// TwinCAT 3 PLC project MainControl
// ProgramVersion: 3.1.4023.0
// libraries:
//   Tc2_EtherCAT, * (Beckhoff Automation GmbH)
//   Tc2_SerialCom, * (Beckhoff Automation GmbH)
//   Tc2_Standard, * (Beckhoff Automation GmbH)
//   Tc2_System, * (Beckhoff Automation GmbH)
//   Tc2_Utilities, * (Beckhoff Automation GmbH)
//   Tc3_EventLogger, * (Beckhoff Automation GmbH)
//   Tc3_Module, * (Beckhoff Automation GmbH)
// project tree:
//   DUTs/ ActivationStatus.TcDUT (not stored), GCControllerMode.TcDUT, GuidanceSystemSTM.TcDUT, HighLevelCondition.TcDUT, LEDColor.TcDUT (not stored), LEDMode.TcDUT (not stored), LevitationSystemSTM.TcDUT (not stored), OperationControlCommands.TcDUT (not stored), TGControllerMode.TcDUT (not stored), TopLevelSTM.TcDUT (not stored), ServiceModuleSTM.TcDUT (not stored), SubLevelCondition.TcDUT, XMCCommands.TcDUT
//   DUTs/Interfaces/ ForwardXMCToOperationControl.TcDUT, FromMainControlToOperationControl.TcDUT, FromMainControlToXMC.TcDUT, FromOperationControlToMainControl.TcDUT (not stored), FromXMCToMainControl.TcDUT
//   GVLs/ OperationControlData.TcGVL, Test.TcGVL, XMCData.TcGVL
//   OOPs/ FB_HighLevelSystem.TcPOU, ITF_HighLevelSystem.TcIO, ITF_SubSystem.TcIO (not stored)
//   POUs/ErrorHandling/ FB_SafetyCounter.TcPOU, FB_EventLogging.TcPOU
//   POUs/ FB_LevitationSystem.TcPOU, PRG_ErrorHandling.TcPOU, PRG_MainController.TcPOU, FB_GuidanceSystem.TcPOU, FB_ServiceModule.TcPOU
//   / PlcTask.TcTTO, PlcTask_Fast.TcTTO
//   POUs/Guidance/AccelerationSensor/ AccelerationSensor.TcGVL, FB_SerialComRS232.TcPOU
//   POUs/Guidance/ FB_AccelerationSensor.TcPOU, FB_GuidanceController.TcPOU
//   POUs/Levitation/ FB_EqualizingController.TcPOU, FB_TrajectoryGenerator.TcPOU
//   POUs/ServiceModule/BoxLED/ BoxLED.TcGVL
//   POUs/ServiceModule/DistanceSensor/ DistanceSensor.TcGVL, FB_SerialComRS422.TcPOU
//   POUs/ServiceModule/ FB_BoxLED.TcPOU, FB_DistanceSensor.TcPOU, FB_RGBLED.TcPOU
//   POUs/ServiceModule/RGBLED/ RGBLED.TcGVL
// real-time tasks:
//   TASK PlcTask: cycle T#1ms, priority 20, ADS port 351
//   TASK PlcTask_Fast: cycle T#1ms, priority 19, ADS port 350
// I/O:
//   DEVICE Gerät 3 (EtherCAT) (disabled), AmsNetId 10.183.66.136.4.1
//     Klemme 1 (EK1100) [EK1100 EtherCAT-Koppler (2A E-Bus)]
//       Klemme 2 (EL6021) [EL6021 Schnittstelle (RS422/485)]
//       Klemme 3 (EL6001) [EL6001 Schnittstelle (RS232)]
//       Klemme 4 (EL6001) [EL6001 Schnittstelle (RS232)]
//       Klemme 5 (EL2564) [EL2564 4 K. LED-Ausgang, 5...48 V DC, 4 A, RGBW]
//       Klemme 6 (EL9011) [EL9011 Endklemme]
//   DEVICE Gerät 4 (EtherCAT Slave) (disabled), AmsNetId 10.183.66.136.5.255
// variable links:
//   MainControl/MainControl Instance <-> Device 3 (EtherCAT)/Term 1 (EK1100)/Term 2 (EL6021)
//     PlcTask Inputs/DistanceSensor.stEL6021In @bit {16..184 step 8} <-> COM TxPDO-Map Inputs/Data In {0..21}  (22 links)
//     PlcTask Inputs/DistanceSensor.stEL6021In <-> COM TxPDO-Map Inputs/Status
//     PlcTask Outputs/DistanceSensor.stEL6021Out <-> COM RxPDO-Map Outputs/Ctrl
//     PlcTask Outputs/DistanceSensor.stEL6021Out @bit {16..184 step 8} <-> COM RxPDO-Map Outputs/Data Out {0..21}  (22 links)
//   MainControl/MainControl Instance <-> Device 3 (EtherCAT)/Term 1 (EK1100)/Term 3 (EL6001)
//     PlcTask Inputs/AccelerationSensor.stEL6001InIMU1 @bit {16..184 step 8} <-> COM Inputs/Data In {0..21}  (22 links)
//     PlcTask Inputs/AccelerationSensor.stEL6001InIMU1 <-> COM Inputs/Status
//     PlcTask Outputs/AccelerationSensor.stEL6001OutIMU1 <-> COM Outputs/Ctrl
//     PlcTask Outputs/AccelerationSensor.stEL6001OutIMU1 @bit {16..184 step 8} <-> COM Outputs/Data Out {0..21}  (22 links)
//   MainControl/MainControl Instance <-> Device 3 (EtherCAT)/Term 1 (EK1100)/Term 4 (EL6001)
//     PlcTask Inputs/AccelerationSensor.stEL6001InIMU2 @bit {16..184 step 8} <-> COM Inputs/Data In {0..21}  (22 links)
//     PlcTask Inputs/AccelerationSensor.stEL6001InIMU2 <-> COM Inputs/Status
//     PlcTask Outputs/AccelerationSensor.stEL6001OutIMU2 <-> COM Outputs/Ctrl
//     PlcTask Outputs/AccelerationSensor.stEL6001OutIMU2 @bit {16..184 step 8} <-> COM Outputs/Data Out {0..21}  (22 links)
//   MainControl/MainControl Instance <-> Device 3 (EtherCAT)/Term 1 (EK1100)/Term 5 (EL2564)
//     PlcTask Inputs/BoxLED.bBoxGreenError <-> PWM Inputs Channel 4/Status/Error
//     PlcTask Inputs/BoxLED.bBoxGreenWarning <-> PWM Inputs Channel 4/Status/Warning
//     PlcTask Outputs/BoxLED.nBoxGreen <-> PWM Outputs Channel 4/PWM output
//   MainControl/MainControl Instance <-> Device 4 (EtherCAT Slave)
//     PlcTask Inputs/OperationControlData.stFromOCToMC <-> Inputs/FromOCToMC
//     PlcTask Outputs/OperationControlData.stForwardXMC{1..4}ToOC <-> Outputs/ForwardXMC{1..4}ToOC  (4 links)
//     PlcTask Outputs/OperationControlData.stFromMCToOC <-> Outputs/FromMCToOC

CONFIGURATION MainControl
    RESOURCE PLC ON TwinCAT3
        TASK PlcTask(INTERVAL := T#1ms, PRIORITY := 20);
        TASK PlcTask_Fast(INTERVAL := T#1ms, PRIORITY := 19);
        PROGRAM PRG_ErrorHandling WITH PlcTask : PRG_ErrorHandling;
        PROGRAM PRG_MainController WITH PlcTask : PRG_MainController;
        PROGRAM PRG_ErrorHandling WITH PlcTask_Fast : PRG_ErrorHandling;
    END_RESOURCE
END_CONFIGURATION

// ---- DUTs/GCControllerMode.TcDUT
{attribute 'qualified_only'}
{attribute 'strict'}
TYPE GCControllerMode :
(
	CurrentControlled,
	ForceControlled
);
END_TYPE

// ---- DUTs/GuidanceSystemSTM.TcDUT
{attribute 'qualified_only'}
{attribute 'strict'}
TYPE GuidanceSystemSTM :
(
	Idling,
	PreRunning,
	Running,
	PostRunning
);
END_TYPE

// ---- DUTs/HighLevelCondition.TcDUT
{attribute 'qualified_only'}
{attribute 'strict'}
TYPE HighLevelCondition :
(
	INIT,
	RUN,
	SLEEP
);
END_TYPE

// ---- DUTs/Interfaces/ForwardXMCToOperationControl.TcDUT
TYPE ForwardXMCToOperationControl :
STRUCT
	MO_origE_State							:	USINT			;
	MO_origE_LoggingCounterIn               :	USINT			;
	MO_origE_LoggingCounterSize             :	USINT			;
	MO_origE_LoggingCounterBuf0             :	BYTE			;
	MO_origE_LoggingCounterBuf1             :	BYTE			;
	MO_origE_LoggingCounterBuf2             :	BYTE			;
	MO_origE_LoggingCounterBuf3             :	BYTE			;
	MO_origE_LoggingCounterBuf4             :	BYTE			;
	MO_origE_LoggingCounterBuf5             :	BYTE			;
	MO_origE_LoggingCounterBuf6             :	BYTE			;
	MO_origE_LoggingCounterBuf7             :	BYTE			;
	MO_origE_LoggingCounterBuf8             :	BYTE			;
	MO_origE_LoggingCounterBuf9             :	BYTE			;
	MO_origE_SafetyCounter                  :	UDINT			;
	MO_origE_Timestamp                      :	UDINT			;
	MO_origE_WarnBits                       :	ULINT			;
	MO_origE_ErrBits                        :	ULINT			;
	MO_origE_DistanceLevitationFiltered     :	REAL			;
	MO_origE_DistanceGuidanceFiltered       :	REAL			;
	MO_origE_DistanceRawLev11               :	REAL			;
	MO_origE_DistanceRawLev12               :	REAL			;
	MO_origE_DistanceRawLev21               :	REAL			;
	MO_origE_DistanceRawLev22               :	REAL			;
	MO_origE_DistanceRawGuid11              :	REAL			;
	MO_origE_DistanceRawGuid12              :	REAL			;
	MO_origE_IMUX                           :	REAL			;
	MO_origE_IMUY                           :	REAL			;
	MO_origE_IMUZ                           :	REAL			;
	MO_origE_VelocityZFiltered              :	REAL			;
	MO_origE_TemperatureBox                 :	REAL			;
	MO_origE_TemperatureLev0                :	REAL			;
	MO_origE_TemperatureLev1                :	REAL			;
	MO_origE_TemperatureGuid                :	REAL			;
	MO_origE_PressureBox                    :	REAL			;
	MO_origE_CurrentLev                     :	DINT			;
	MO_origE_CurrentGuid                    :	DINT			;
	MO_origE_GuidEstimatedFlux0             :	ARRAY [0..1] OF REAL			;
	MO_origE_GuidEstimatedFlux1             :	ARRAY [0..1] OF REAL			;
	MO_origE_GuidEstimatedCurrent           :	REAL			;
	MO_origE_GuidEstimatedResistance        :	REAL			;
	MO_origE_GuidIntegratedControlError     :	REAL			;
	MO_origE_GuidReferenceVoltage           :	REAL			;
	MO_origE_LevEstimatedFlux0              :	ARRAY [0..1] OF REAL			;
	MO_origE_LevEstimatedFlux1              :	ARRAY [0..1] OF REAL			;
	MO_origE_LevEstimatedCurrent            :	REAL			;
	MO_origE_LevEstimatedResistance         :	REAL			;
	MO_origE_LevIntegratedControlError      :	REAL			;
	MO_origE_LevReferenceVoltage            :	REAL			;
END_STRUCT
END_TYPE

// ---- DUTs/Interfaces/FromMainControlToOperationControl.TcDUT
TYPE FromMainControlToOperationControl :
STRUCT
		//MainController
		MO_origM_State 							: USINT		;
		MO_origM_WarnBits 						: ULINT		;
		MO_origM_ErrBits 						: ULINT		;
		MO_origM_SafetyCounter 					: UDINT		;
		MO_origM_ShutdownFinished 				: BIT		;
		//ServiceModule                 		
		MO_origM_DistanceServiceModule 			: REAL		;
		
		//LevitationSystem
		MO_origM_ECOutputDistanceXMC1 			: REAL		;
		MO_origM_ECOutputDistanceXMC2 			: REAL		;
		MO_origM_ECOutputDistanceXMC3 			: REAL		;
		MO_origM_ECOutputDistanceXMC4 			: REAL		;
		MO_origM_TGOutputLevDistanceXMC1 		: REAL		;
		MO_origM_TGOutputLevDistanceXMC2 		: REAL		;
		MO_origM_TGOutputLevDistanceXMC3 		: REAL		;
		MO_origM_TGOutputLevDistanceXMC4 		: REAL		;
		MO_origM_TGOutputLevVelocityXMC1 		: REAL		;
		MO_origM_TGOutputLevVelocityXMC2 		: REAL		;
		MO_origM_TGOutputLevVelocityXMC3 		: REAL		;
		MO_origM_TGOutputLevVelocityXMC4 		: REAL		;
		MO_origM_TGOutputLevAccelerationXMC1 	: REAL		;
		MO_origM_TGOutputLevAccelerationXMC2 	: REAL		;
		MO_origM_TGOutputLevAccelerationXMC3 	: REAL		;
		MO_origM_TGOutputLevAccelerationXMC4 	: REAL		;
		MO_origM_TGOutputLevCurrentXMC1 		: REAL		;
		MO_origM_TGOutputLevCurrentXMC2 		: REAL		;
		MO_origM_TGOutputLevCurrentXMC3 		: REAL		;
		MO_origM_TGOutputLevCurrentXMC4 		: REAL		;
		MO_origM_TGOutputLevVoltageXMC1 		: REAL		;
		MO_origM_TGOutputLevVoltageXMC2 		: REAL		;
		MO_origM_TGOutputLevVoltageXMC3 		: REAL		;
		MO_origM_TGOutputLevVoltageXMC4 		: REAL		;
		MO_origM_TGOutputLevForceXMC1 			: REAL		;
		MO_origM_TGOutputLevForceXMC2 			: REAL		;
		MO_origM_TGOutputLevForceXMC3 			: REAL		;
		MO_origM_TGOutputLevForceXMC4 			: REAL		;
		
		//GuidanceSystem
		MO_origM_GuidanceIMUX0 					: REAL		;
		MO_origM_GuidanceIMUX1 					: REAL		;
		MO_origM_GuidanceIMUY0 					: REAL		;
		MO_origM_GuidanceIMUY1 					: REAL		;
		MO_origM_GuidanceIMUZ0 					: REAL		;
		MO_origM_GuidanceIMUZ1 					: REAL		;
		MO_origM_GCOutputGuidCurrentXMC1 		: REAL		;
		MO_origM_GCOutputGuidCurrentXMC2 		: REAL		;
		MO_origM_GCOutputGuidCurrentXMC3 		: REAL		;
		MO_origM_GCOutputGuidCurrentXMC4 		: REAL		;
		MO_origM_GCOutputGuidVoltageXMC1 		: REAL		;
		MO_origM_GCOutputGuidVoltageXMC2 		: REAL		;
		MO_origM_GCOutputGuidVoltageXMC3 		: REAL		;
		MO_origM_GCOutputGuidVoltageXMC4 		: REAL		;
		MO_origM_GCOutputGuidForceXMC1 			: REAL		;
		MO_origM_GCOutputGuidForceXMC2 			: REAL		;
		MO_origM_GCOutputGuidForceXMC3 			: REAL		;
		MO_origM_GCOutputGuidForceXMC4 			: REAL		;
END_STRUCT
END_TYPE

// ---- DUTs/Interfaces/FromMainControlToXMC.TcDUT
TYPE FromMainControlToXMC :
STRUCT
	ME_origM_StartOperational						:	BIT		;
	ME_origM_StopOperational                        :	BIT    	;
	ME_origM_AckError                               :	BIT    	;
	ME_origG_Logging_CounterOut                     :	USINT   ;
	ME_origM_SafetyCounter                          :	UDINT   ;
	ME_origM_DesiredGuidCurrent                     :	REAL    ;
	ME_origM_DesiredGuidForce                       :	REAL    ;
	ME_origM_DesiredGuidVoltage                     :	REAL    ;
	ME_origM_DesiredLevDistance                     :	REAL    ;
	ME_origM_DesiredLevVelocity                     :	REAL    ;
	ME_origM_DesiredLevAcceleration                 :	REAL    ;
	ME_origM_DesiredLevForce                        :	REAL    ;
	ME_origM_DesiredLevCurrent                      :	REAL    ;
	ME_origM_DesiredLevVoltage                      :	REAL    ;
	ME_origM_DebugPWMLev                            :	INT     ;
	ME_origM_DebugPWMGuid                           :	INT     ;
	ME_origM_DebugSel                               :	USINT   ;
	ME_origG_GuidControlOption                      :	USINT   ;
	ME_origG_LevControlOption                       :	USINT   ;
	ME_origG_EnableGuidController                   :	BIT    	;
	ME_origM_GuidEnableCurrentController            :	BIT    	;
	ME_origM_GuidEnableIControl                     :	BIT    	;
	ME_origM_GuidEnablePControl                     :	BIT    	;
	ME_origM_LevEnableCurrentController             :	BIT    	;
	ME_origM_LevEnableIControl                      :	BIT    	;
	ME_origM_LevEnablePControl                      :	BIT    	;
END_STRUCT
END_TYPE

// ---- DUTs/Interfaces/FromXMCToMainControl.TcDUT
TYPE FromXMCToMainControl :
STRUCT
	EM_origE_State							:	USINT			;
	EM_origE_LoggingCounterIn               :	USINT			;
	EM_origE_LoggingCounterSize             :	USINT			;
	EM_origE_LoggingCounterBuf0             :	BYTE			;
	EM_origE_LoggingCounterBuf1             :	BYTE			;
	EM_origE_LoggingCounterBuf2             :	BYTE			;
	EM_origE_LoggingCounterBuf3             :	BYTE			;
	EM_origE_LoggingCounterBuf4             :	BYTE			;
	EM_origE_LoggingCounterBuf5             :	BYTE			;
	EM_origE_LoggingCounterBuf6             :	BYTE			;
	EM_origE_LoggingCounterBuf7             :	BYTE			;
	EM_origE_LoggingCounterBuf8             :	BYTE			;
	EM_origE_LoggingCounterBuf9             :	BYTE			;
	EM_origE_SafetyCounter                  :	UDINT			;
	EM_origE_Timestamp                      :	UDINT			;
	EM_origE_WarnBits                       :	ULINT			;
	EM_origE_ErrBits                        :	ULINT			;
	EM_origE_DistanceLevitationFiltered     :	REAL			;
	EM_origE_DistanceGuidanceFiltered       :	REAL			;
	EM_origE_DistanceRawLev11               :	REAL			;
	EM_origE_DistanceRawLev12               :	REAL			;
	EM_origE_DistanceRawLev21               :	REAL			;
	EM_origE_DistanceRawLev22               :	REAL			;
	EM_origE_DistanceRawGuid11              :	REAL			;
	EM_origE_DistanceRawGuid12              :	REAL			;
	EM_origE_IMUX                           :	REAL			;
	EM_origE_IMUY                           :	REAL			;
	EM_origE_IMUZ                           :	REAL			;
	EM_origE_VelocityZFiltered              :	REAL			;
	EM_origE_TemperatureBox                 :	REAL			;
	EM_origE_TemperatureLev0                :	REAL			;
	EM_origE_TemperatureLev1                :	REAL			;
	EM_origE_TemperatureGuid                :	REAL			;
	EM_origE_PressureBox                    :	REAL			;
	EM_origE_CurrentLev                     :	DINT			;
	EM_origE_CurrentGuid                    :	DINT			;
	EM_origE_GuidEstimatedFlux0             :	ARRAY [0..1] OF REAL;
	EM_origE_GuidEstimatedFlux1             :	ARRAY [0..1] OF REAL			;
	EM_origE_GuidEstimatedCurrent           :	REAL			;
	EM_origE_GuidEstimatedResistance        :	REAL			;
	EM_origE_GuidIntegratedControlError     :	REAL			;
	EM_origE_GuidReferenceVoltage           :	REAL			;
	EM_origE_LevEstimatedFlux0              :	ARRAY [0..1] OF REAL			;
	EM_origE_LevEstimatedFlux1              :	ARRAY [0..1] OF REAL			;
	EM_origE_LevEstimatedCurrent            :	REAL			;
	EM_origE_LevEstimatedResistance         :	REAL			;
	EM_origE_LevIntegratedControlError      :	REAL			;
	EM_origE_LevReferenceVoltage            :	REAL			;
END_STRUCT
END_TYPE

// ---- DUTs/SubLevelCondition.TcDUT
{attribute 'qualified_only'}
{attribute 'strict'}
TYPE SubLevelCondition :
(
	ERROR,
	RUN
);
END_TYPE

// ---- DUTs/XMCCommands.TcDUT
TYPE XMCCommands :
STRUCT
	//MainController
	nSafetyCounterXMC1 			: UDINT	;
	nSafetyCounterXMC2 			: UDINT	;
	nSafetyCounterXMC3 			: UDINT	;
	nSafetyCounterXMC4 			: UDINT	;
	nStateXMC1					: USINT	;
	nStateXMC2					: USINT	;
	nStateXMC3					: USINT	;
	nStateXMC4					: USINT	;
	
	//Outputs
	bStartOperational : BOOL;
	bStopOperational	: BOOL;
	bAckError			: BOOL;
	nDebugPWMSel		: USINT;
	nDebugPWMLev		: INT;
	nDebugPWMGuid		: INT;
END_STRUCT
END_TYPE

// ---- GVLs/OperationControlData.TcGVL
{attribute 'qualified_only'}
VAR_GLOBAL
	stFromOCToMC 			AT %I* : FromOperationControlToMainControl;
	
	stFromMCToOC 			AT %Q* : FromMainControlToOperationControl;
	stForwardXMC1ToOC 		AT %Q* : ForwardXMCToOperationControl;
	stForwardXMC2ToOC 		AT %Q* : ForwardXMCToOperationControl;
	stForwardXMC3ToOC 		AT %Q* : ForwardXMCToOperationControl;
	stForwardXMC4ToOC 		AT %Q* : ForwardXMCToOperationControl;
END_VAR

// ---- GVLs/Test.TcGVL
{attribute 'qualified_only'}
VAR_GLOBAL
	nTest AT %Q* : INT;
END_VAR

// ---- GVLs/XMCData.TcGVL
{attribute 'qualified_only'}
VAR_GLOBAL
	stFromXMC1ToMC 			AT %I* : FromXMCToMainControl;
	stFromXMC2ToMC 			AT %I* : FromXMCToMainControl;
	stFromXMC3ToMC 			AT %I* : FromXMCToMainControl;
	stFromXMC4ToMC 			AT %I* : FromXMCToMainControl;
	
	stFromMCToXMC1			AT %Q* : FromMainControlToXMC;
	stFromMCToXMC2			AT %Q* : FromMainControlToXMC;
	stFromMCToXMC3			AT %Q* : FromMainControlToXMC;
	stFromMCToXMC4			AT %Q* : FromMainControlToXMC;
END_VAR

// ---- POUs/Guidance/AccelerationSensor/AccelerationSensor.TcGVL
VAR_GLOBAL
	stEL6001InIMU1 AT %I*	: EL6inData22B;		//**To EL6001 Inputs incl. Status (Clamp 3)**
	stEL6001OutIMU1 AT %Q*	: EL6outData22B;	//**To EL6001 Outputs incl. Ctrl (Clamp 3)**
	
	stEL6001InIMU2 AT %I*	: EL6inData22B;		//**To EL6001 Inputs incl. Status (Clamp 4)**
	stEL6001OutIMU2 AT %Q*	: EL6outData22B;	//**To EL6001 Outputs incl. Ctrl (Clamp 4)** 
END_VAR

// ---- POUs/ServiceModule/BoxLED/BoxLED.TcGVL
{attribute 'qualified_only'}
VAR_GLOBAL
	nBoxGreen AT %Q* : INT;					//**To EL2564 PWM Outputs Channel 4 (PWM output)**
	
	bBoxGreenError AT %I* : BOOL;				//**To EL2564 PWM Inputs Channel 4 (Status -> Error)**
	bBoxGreenWarning AT %I* : BOOL;			//**To EL2564 PWM Inputs Channel 4 (Status -> Warning)**
END_VAR

// ---- POUs/ServiceModule/DistanceSensor/DistanceSensor.TcGVL
{attribute 'qualified_only'}
VAR_GLOBAL
	stEL6021In  AT %I*	: EL6inData22B;		//**To EL6021 Inputs**
	stEL6021Out AT %Q*	: EL6outData22B;	//**To EL6021 Outputs**
END_VAR

// ---- POUs/ServiceModule/RGBLED/RGBLED.TcGVL
{attribute 'qualified_only'}
VAR_GLOBAL
	nRed AT %Q* : INT;				//**To EL2564 PWM Outputs Channel 1 (PWM output)**
	nGreen AT %Q* : INT;			//**To EL2564 PWM Outputs Channel 2 (PWM output)**
	nBlue AT %Q* : INT;				//**To EL2564 PWM Outputs Channel 3 (PWM output)**
	
	bRedError AT %I* : BOOL;		//**To EL2564 PWM Inputs Channel 1 (Status -> Error)**
	bRedWarning AT %I* : BOOL;		//**To EL2564 PWM Inputs Channel 1 (Status -> Warning)**
	bGreenError AT %I* : BOOL;		//**To EL2564 PWM Inputs Channel 2 (Status -> Error)**
	bGreenWarning AT %I* : BOOL;	//**To EL2564 PWM Inputs Channel 2 (Status -> Warning)**
	bBlueError AT %I* : BOOL;		//**To EL2564 PWM Inputs Channel 3 (Status -> Error)**
	bBlueWarning AT %I* : BOOL;		//**To EL2564 PWM Inputs Channel 3 (Status -> Warning)**
END_VAR

// ---- OOPs/ITF_HighLevelSystem.TcIO
INTERFACE ITF_HighLevelSystem

PROPERTY PUBLIC eCondition : HighLevelCondition
GET
END_GET
END_PROPERTY

PROPERTY PUBLIC nErrorID : UDINT
GET
END_GET
END_PROPERTY

END_INTERFACE

// ---- POUs/PRG_ErrorHandling.TcPOU
PROGRAM PRG_ErrorHandling
VAR
	nErrorBits 						: ULINT;
	nWarningBits 					: ULINT;
	
	fbStartUpTimer 					: TON := (PT := tStartUpTime);
	fbShutdownTimer					: TON := (PT := tShutdownTime);
	bStartUpCheck 					: BOOL;
	bErrorInStartUp 				: BOOL;
	bErrorInReady 					: BOOL;
	bErrorInOperational 			: BOOL;
	bErrorInShutdown 				: BOOL;
	bGoToError						: BOOL;
	bAllErrorsAcknowledged 			: BOOL;
	
	fbEventLogging 					: FB_EventLogging;
	aSetEventCounterToZero 			: ARRAY [0..nNumberOfWarnings + nNumberOfErrors + nNumberOfInfos - 1] OF USINT;
	n 								: USINT;
	
	fbSafetyCounter 				: FB_SafetyCounter;
	
	bDebugMode 						: BOOL;
	nTestMode						: USINT := 63;  //*see test modes table in README*
END_VAR
VAR CONSTANT
	tStartUpTime 					: TIME := T#10S;
	tSafetyCounterTimeout 			: TIME := T#5S;
	tShutdownTime					: TIME := T#30S;
	
	nNumberOfWarnings 				: USINT := 52;			//*set the number of Warnings here*
	nNumberOfErrors 				: USINT := 6;			//*set the number of Errors here*
	nNumberOfInfos					: USINT := 4;			//*set the number of Infos here*
END_VAR

doSetWarningBits(	nErrorIDServiceModule := PRG_MainController.fbServiceModule.nErrorID,
					nErrorIDLevitationSystem := PRG_MainController.fbLevitationSystem.nErrorID,
					nErrorIDGuidanceSystem := PRG_MainController.fbGuidanceSystem.nErrorID,
					nErrorIDMainController := PRG_ErrorHandling.fbSafetyCounter.nErrorID);
					
doSetErrorBits(		nErrorIDServiceModule := PRG_MainController.fbServiceModule.nErrorID,
					nErrorIDLevitationSystem := PRG_MainController.fbLevitationSystem.nErrorID,
					nErrorIDGuidanceSystem := PRG_MainController.fbGuidanceSystem.nErrorID,
					nErrorIDMainController := PRG_ErrorHandling.fbSafetyCounter.nErrorID);

doCheckErrorStates();

fbSafetyCounter();
fbEventLogging();

IF bDebugMode THEN
	nErrorBits := 0;
END_IF

							
CASE PRG_MainController.eState OF
	TopLevelSTM.STARTUP:
		bAllErrorsAcknowledged := FALSE;
		
		IF NOT bDebugMode AND NOT nTestMode.1 THEN
			doStartUpCheck(	eConditionServiceModule := PRG_MainController.fbServiceModule.eCondition,
							eConditionLevitationSystem := PRG_MainController.fbLevitationSystem.eCondition,
							eConditionGuidanceSystem := PRG_MainController.fbGuidanceSystem.eCondition);
		ELSE
			bStartUpCheck := TRUE;
		END_IF	
										
	TopLevelSTM.READY:
		fbShutdownTimer(IN:=FALSE);
		IF nErrorBits <> 0 THEN
			bErrorInReady := TRUE;
		ELSE
			bErrorInReady := FALSE;
		END_IF
		
	TopLevelSTM.OPERATIONAL:
		IF nErrorBits <> 0 THEN
			bErrorInOperational := TRUE;
		ELSE
			bErrorInOperational := FALSE;
		END_IF
		
	TopLevelSTM.SHUTDOWN:
		fbShutdownTimer(IN:=TRUE);
		IF NOT bErrorInOperational THEN
			IF nErrorBits <> 0 THEN
				bErrorInShutdown := TRUE;
			ELSE
				bErrorInShutdown := FALSE;
			END_IF
		END_IF
		
	TopLevelSTM.ERROR:
		IF PRG_MainController.stOperationControlCommands.bAckError THEN
			
			//Reset WarningBits and ErrorBits
			nWarningBits := 0;
			nErrorBits := 0;
			
			//Reset Event Logging
			FOR n := 0 TO nNumberOfWarnings + nNumberOfErrors + nNumberOfInfos -1 DO
				aSetEventCounterToZero[n] := 0;
			END_FOR
			fbEventLogging.aEventCounter := aSetEventCounterToZero;
			
			//ResetSafetyCounter
			fbSafetyCounter(bReset := TRUE);
			fbSafetyCounter.bReset := FALSE;
			
			//Acknowledge
			bErrorInStartUp := FALSE;
			bErrorInReady := FALSE;
			bErrorInOperational := FALSE;
			bErrorInShutdown := FALSE;
			bAllErrorsAcknowledged := TRUE;
		END_IF
END_CASE

METHOD PRIVATE doCheckErrorStates
IF PRG_MainController.stXMCCommands.nStateXMC1 = 3 OR PRG_MainController.stXMCCommands.nStateXMC2 = 3 OR PRG_MainController.stXMCCommands.nStateXMC3 = 3 OR PRG_MainController.stXMCCommands.nStateXMC4 = 3 OR PRG_MainController.stOperationControlCommands.bGoToError THEN
	bGoToError := TRUE;
ELSE
	bGoToError := FALSE;
END_IF
END_METHOD

METHOD PRIVATE doSetErrorBits
VAR_INPUT
	nErrorIDServiceModule : UDINT;
	nErrorIDLevitationSystem : UDINT;
	nErrorIDGuidanceSystem : UDINT;
	nErrorIDMainController : UDINT;
END_VAR
IF PRG_MainController.fbServiceModule.eActivationStatus = ActivationStatus.Disabled THEN
	nErrorIDServiceModule := 0;
END_IF
IF PRG_MainController.fbLevitationSystem.eActivationStatus = ActivationStatus.Disabled THEN
	nErrorIDLevitationSystem := 0;
	nErrorIDMainController.1 := 0;
	nErrorIDMainController.2 := 0;
	nErrorIDMainController.3 := 0;
	nErrorIDMainController.4 := 0;
END_IF
IF PRG_MainController.fbGuidanceSystem.eActivationStatus = ActivationStatus.Disabled THEN
	nErrorIDGuidanceSystem := 0;
	nErrorIDMainController.1 := 0;
	nErrorIDMainController.2 := 0;
	nErrorIDMainController.3 := 0;
	nErrorIDMainController.4 := 0;
END_IF


//ServiceModule

//LevitationSystem

//GuidanceSystem
		
//MainController
nErrorBits.0 := nErrorIDMainController.0;
nErrorBits.1 := nErrorIDMainController.1;
nErrorBits.2 := nErrorIDMainController.2;
nErrorBits.3 := nErrorIDMainController.3;
nErrorBits.4 := nErrorIDMainController.4;
nErrorBits.5 := nErrorIDMainController.5;
END_METHOD

METHOD PRIVATE doSetWarningBits
VAR_INPUT
	nErrorIDServiceModule : UDINT;
	nErrorIDLevitationSystem : UDINT;
	nErrorIDGuidanceSystem : UDINT;
	nErrorIDMainController : UDINT;
END_VAR
IF PRG_MainController.fbServiceModule.eActivationStatus = ActivationStatus.Disabled THEN
	nErrorIDServiceModule := 0;
END_IF
IF PRG_MainController.fbLevitationSystem.eActivationStatus = ActivationStatus.Disabled THEN
	nErrorIDLevitationSystem := 0;
END_IF
IF PRG_MainController.fbGuidanceSystem.eActivationStatus = ActivationStatus.Disabled THEN
	nErrorIDGuidanceSystem := 0;
END_IF

//ServiceModule
nWarningBits.0 := nErrorIDServiceModule.0;
nWarningBits.1 := nErrorIDServiceModule.1;
nWarningBits.2 := nErrorIDServiceModule.2;
nWarningBits.3 := nErrorIDServiceModule.3;
nWarningBits.4 := nErrorIDServiceModule.4;
nWarningBits.5 := nErrorIDServiceModule.5;
nWarningBits.6 := nErrorIDServiceModule.6;
nWarningBits.7 := nErrorIDServiceModule.7;
nWarningBits.8 := nErrorIDServiceModule.8;
nWarningBits.9 := nErrorIDServiceModule.9;

//LevitationSystem
nWarningBits.10 := nErrorIDLevitationSystem.0;
nWarningBits.11 := nErrorIDLevitationSystem.1;
nWarningBits.12 := nErrorIDLevitationSystem.2;
nWarningBits.13 := nErrorIDLevitationSystem.3;
nWarningBits.14 := nErrorIDLevitationSystem.4;
nWarningBits.15 := nErrorIDLevitationSystem.5;
nWarningBits.16 := nErrorIDLevitationSystem.6;
nWarningBits.17 := nErrorIDLevitationSystem.7;
nWarningBits.18 := nErrorIDLevitationSystem.8;
nWarningBits.19 := nErrorIDLevitationSystem.9;
nWarningBits.20 := nErrorIDLevitationSystem.10;
nWarningBits.21 := nErrorIDLevitationSystem.11;
nWarningBits.22 := nErrorIDLevitationSystem.12;
nWarningBits.23 := nErrorIDLevitationSystem.13;
nWarningBits.24 := nErrorIDLevitationSystem.14;
nWarningBits.25 := nErrorIDLevitationSystem.15;
nWarningBits.26 := nErrorIDLevitationSystem.16;
nWarningBits.27 := nErrorIDLevitationSystem.17;
nWarningBits.28 := nErrorIDLevitationSystem.18;
nWarningBits.29 := nErrorIDLevitationSystem.19;
nWarningBits.30 := nErrorIDLevitationSystem.20;
nWarningBits.31 := nErrorIDLevitationSystem.21;
nWarningBits.32 := nErrorIDLevitationSystem.22;
nWarningBits.33 := nErrorIDLevitationSystem.23;
nWarningBits.34 := nErrorIDLevitationSystem.24;
nWarningBits.35 := nErrorIDLevitationSystem.25;


//GuidanceSystem
nWarningBits.36 := nErrorIDGuidanceSystem.0;
nWarningBits.37 := nErrorIDGuidanceSystem.1;
nWarningBits.38 := nErrorIDGuidanceSystem.2;
nWarningBits.39 := nErrorIDGuidanceSystem.3;
nWarningBits.40 := nErrorIDGuidanceSystem.4;
nWarningBits.41 := nErrorIDGuidanceSystem.5;
nWarningBits.42 := nErrorIDGuidanceSystem.6;
nWarningBits.43 := nErrorIDGuidanceSystem.7;
nWarningBits.44 := nErrorIDGuidanceSystem.8;
nWarningBits.45 := nErrorIDGuidanceSystem.9;
nWarningBits.46 := nErrorIDGuidanceSystem.10;
nWarningBits.47 := nErrorIDGuidanceSystem.11;
nWarningBits.48 := nErrorIDGuidanceSystem.12;
nWarningBits.49 := nErrorIDGuidanceSystem.13;
nWarningBits.50 := nErrorIDGuidanceSystem.14;
nWarningBits.51 := nErrorIDGuidanceSystem.15;

//MainController
END_METHOD

METHOD PRIVATE doStartUpCheck
VAR_INPUT
	eConditionServiceModule : HighLevelCondition;
	eConditionLevitationSystem : HighLevelCondition;
	eConditionGuidanceSystem : HighLevelCondition;
END_VAR
IF PRG_MainController.stOperationControlCommands.nOperationMode <> 7 THEN
	IF (eConditionServiceModule = HighLevelCondition.RUN OR eConditionServiceModule = HighLevelCondition.SLEEP) AND (eConditionLevitationSystem = HighLevelCondition.RUN OR eConditionLevitationSystem = HighLevelCondition.SLEEP) AND (eConditionGuidanceSystem = HighLevelCondition.RUN OR eConditionGuidanceSystem = HighLevelCondition.SLEEP) AND NOT (eConditionServiceModule = HighLevelCondition.SLEEP AND eConditionLevitationSystem = HighLevelCondition.SLEEP AND eConditionGuidanceSystem = HighLevelCondition.SLEEP) THEN
		fbStartUpTimer(IN := FALSE);
		bStartUpCheck := TRUE;
	ELSE
		fbStartUpTimer(IN := TRUE);
		IF fbStartUpTimer.Q THEN
			fbStartUpTimer(IN := FALSE);
			bErrorInStartUp := TRUE;
			bStartUpCheck := FALSE;
		ELSE
			bStartUpCheck := FALSE;
		END_IF
	END_IF
ELSE
		fbStartUpTimer(IN := TRUE);
		IF fbStartUpTimer.Q THEN
			fbStartUpTimer(IN := FALSE);
			bErrorInStartUp := TRUE;
			bStartUpCheck := FALSE;
		ELSE
			bStartUpCheck := FALSE;
		END_IF
END_IF
END_METHOD

END_PROGRAM

// ---- POUs/ErrorHandling/FB_EventLogging.TcPOU
FUNCTION_BLOCK FB_EventLogging
VAR
	fbEventMessage : FB_TcMessage;
	fbEventLogger : FB_TcEventLogger;
	fbCsvExport : FB_TcEventCsvExportSettings;
	fbCsvClear : FB_TcClearLoggedEventsSettings;

	
	n : USINT;
	aCounterID : ARRAY [0..PRG_ErrorHandling.nNumberOfWarnings + PRG_ErrorHandling.nNumberOfErrors + PRG_ErrorHandling.nNumberOfInfos - 1] OF USINT;
	aWarningArray : ARRAY [0..PRG_ErrorHandling.nNumberOfWarnings-1] OF BOOL;
	aWarningMessagesAsStrings : ARRAY [0..PRG_ErrorHandling.nNumberOfWarnings-1] OF STRING;
	aErrorArray : ARRAY [0..PRG_ErrorHandling.nNumberOfErrors-1] OF BOOL;
	aErrorMessagesAsStrings : ARRAY [0..PRG_ErrorHandling.nNumberOfErrors-1] OF STRING;
	aInfoArray : ARRAY [0..PRG_ErrorHandling.nNumberOfInfos-1] OF BOOL;
	aInfoMessagesAsStrings : ARRAY [0..PRG_ErrorHandling.nNumberOfInfos - 1] OF STRING;
	eMainControllerState : TopLevelSTM;
	sMainControllerStateAsString : STRING;
	
	bClearLoggedEvents : BOOL;
	fbExportTimer : TON;
END_VAR
VAR CONSTANT
	nCounterMax : USINT := 255; //max value for USINT data type
	nCounterReset : USINT := 2;
END_VAR

//CSV-Export
fbExportTimer(IN:=TRUE, PT:=T#5S);
IF fbExportTimer.Q THEN
	fbEventLogger.ExportLoggedEvents(sFileName:='C:\Users\Administrator\Desktop\Log.csv', ipExportSettings := fbCsvExport);
	fbExportTimer(IN := FALSE);
END_IF
//CSV-Clear
IF bClearLoggedEvents THEN
	fbEventLogger.ClearLoggedEvents(ipClearSettings:=fbCsvClear);	
END_IF

//TransitionLogging
sMainControllerStateAsString := TO_STRING(PRG_MainController.eState);
IF eMainControllerState <> PRG_MainController.eState THEN
	eMainControllerState := PRG_MainController.eState; 
	fbEventMessage.CreateEx(stEventEntry:=TC_Events.MainControlEventClass.STMTransition, 0);
	fbEventMessage.ipArguments.AddString('MainController').AddString(sMainControllerStateAsString);
	fbEventMessage.Send(0);
END_IF

//InfoMessages
//*Add New Info Messages Here*
aInfoArray[0] := PRG_ErrorHandling.bAllErrorsAcknowledged;
aInfoArray[1] := (NOT TO_BOOL(PRG_MainController.fbServiceModule.eActivationStatus) AND PRG_MainController.stOperationControlCommands.nOperationMode.0);
aInfoArray[2] := (NOT TO_BOOL(PRG_MainController.fbLevitationSystem.eActivationStatus) AND PRG_MainController.stOperationControlCommands.nOperationMode.1);
aInfoArray[3] := (NOT TO_BOOL(PRG_MainController.fbGuidanceSystem.eActivationStatus) AND PRG_MainController.stOperationControlCommands.nOperationMode.2);

aInfoMessagesAsStrings[0] := 'All Errors Acknowledged and Cleared by Operation Control';
aInfoMessagesAsStrings[1] := 'Service Module disabled';
aInfoMessagesAsStrings[2] := 'Levitation System disabled';
aInfoMessagesAsStrings[3] := 'Guidance System disabled';

FOR n := 0 TO PRG_ErrorHandling.nNumberOfInfos-1 DO
	IF aInfoArray[n] THEN
		aCounterID[n + PRG_ErrorHandling.nNumberOfWarnings + PRG_ErrorHandling.nNumberOfErrors] := aCounterID[n + PRG_ErrorHandling.nNumberOfWarnings + PRG_ErrorHandling.nNumberOfErrors] + 1;
		IF aCounterID[n + PRG_ErrorHandling.nNumberOfWarnings + PRG_ErrorHandling.nNumberOfErrors] = nCounterMax THEN
			aCounterID[n + PRG_ErrorHandling.nNumberOfWarnings + PRG_ErrorHandling.nNumberOfErrors] := nCounterReset;
		END_IF
		fbEventMessage.CreateEx(stEventEntry:=TC_Events.MainControlEventClass.Info, 0);
		IF aCounterID[n + PRG_ErrorHandling.nNumberOfWarnings + PRG_ErrorHandling.nNumberOfErrors] = 1 THEN
			fbEventMessage.ipArguments.Clear().AddString(aInfoMessagesAsStrings[n]);
			fbEventMessage.Send(0);
		END_IF
	ELSE
		aCounterID[n + PRG_ErrorHandling.nNumberOfWarnings + PRG_ErrorHandling.nNumberOfErrors] := 0;
	END_IF	
END_FOR

//WarningMessages
//*Add New Warning Messages Here*
aWarningArray[0] := PRG_ErrorHandling.nWarningBits.0;
aWarningArray[1] := PRG_ErrorHandling.nWarningBits.1;
aWarningArray[2] := PRG_ErrorHandling.nWarningBits.2;
aWarningArray[3] := PRG_ErrorHandling.nWarningBits.3;
aWarningArray[4] := PRG_ErrorHandling.nWarningBits.4;
aWarningArray[5] := PRG_ErrorHandling.nWarningBits.5;
aWarningArray[6] := PRG_ErrorHandling.nWarningBits.6;
aWarningArray[7] := PRG_ErrorHandling.nWarningBits.7;
aWarningArray[8] := PRG_ErrorHandling.nWarningBits.8;
aWarningArray[9] := PRG_ErrorHandling.nWarningBits.9;
aWarningArray[10] := PRG_ErrorHandling.nWarningBits.10;
aWarningArray[11] := PRG_ErrorHandling.nWarningBits.11;
aWarningArray[12] := PRG_ErrorHandling.nWarningBits.12;
aWarningArray[13] := PRG_ErrorHandling.nWarningBits.13;
aWarningArray[14] := PRG_ErrorHandling.nWarningBits.14;
aWarningArray[15] := PRG_ErrorHandling.nWarningBits.15;
aWarningArray[16] := PRG_ErrorHandling.nWarningBits.16;
aWarningArray[17] := PRG_ErrorHandling.nWarningBits.17;
aWarningArray[18] := PRG_ErrorHandling.nWarningBits.18;
aWarningArray[19] := PRG_ErrorHandling.nWarningBits.19;
aWarningArray[20] := PRG_ErrorHandling.nWarningBits.20;
aWarningArray[21] := PRG_ErrorHandling.nWarningBits.21;
aWarningArray[22] := PRG_ErrorHandling.nWarningBits.22;
aWarningArray[23] := PRG_ErrorHandling.nWarningBits.23;
aWarningArray[24] := PRG_ErrorHandling.nWarningBits.24;
aWarningArray[25] := PRG_ErrorHandling.nWarningBits.25;
aWarningArray[26] := PRG_ErrorHandling.nWarningBits.26;
aWarningArray[27] := PRG_ErrorHandling.nWarningBits.27;
aWarningArray[28] := PRG_ErrorHandling.nWarningBits.28;
aWarningArray[29] := PRG_ErrorHandling.nWarningBits.29;
aWarningArray[30] := PRG_ErrorHandling.nWarningBits.30;
aWarningArray[31] := PRG_ErrorHandling.nWarningBits.31;
aWarningArray[32] := PRG_ErrorHandling.nWarningBits.32;
aWarningArray[33] := PRG_ErrorHandling.nWarningBits.33;
aWarningArray[34] := PRG_ErrorHandling.nWarningBits.34;
aWarningArray[35] := PRG_ErrorHandling.nWarningBits.35;
aWarningArray[36] := PRG_ErrorHandling.nWarningBits.36;
aWarningArray[37] := PRG_ErrorHandling.nWarningBits.37;
aWarningArray[38] := PRG_ErrorHandling.nWarningBits.38;
aWarningArray[39] := PRG_ErrorHandling.nWarningBits.39;
aWarningArray[40] := PRG_ErrorHandling.nWarningBits.40;
aWarningArray[41] := PRG_ErrorHandling.nWarningBits.41;
aWarningArray[42] := PRG_ErrorHandling.nWarningBits.42;
aWarningArray[43] := PRG_ErrorHandling.nWarningBits.43;
aWarningArray[44] := PRG_ErrorHandling.nWarningBits.44;
aWarningArray[45] := PRG_ErrorHandling.nWarningBits.45;
aWarningArray[46] := PRG_ErrorHandling.nWarningBits.46;
aWarningArray[47] := PRG_ErrorHandling.nWarningBits.47;
aWarningArray[48] := PRG_ErrorHandling.nWarningBits.48;
aWarningArray[49] := PRG_ErrorHandling.nWarningBits.49;
aWarningArray[50] := PRG_ErrorHandling.nWarningBits.50;
aWarningArray[51] := PRG_ErrorHandling.nWarningBits.51;		

aWarningMessagesAsStrings[0] :=		'DistanceSensor Communication Error					';      
aWarningMessagesAsStrings[1] :=    	'DistanceSensor out of Range						';             
aWarningMessagesAsStrings[2] :=    	'BoxLED Temperature too high						';             
aWarningMessagesAsStrings[3] :=    	'BoxLED No Supply Voltage							';                
aWarningMessagesAsStrings[4] :=    	'RedLED Temperature too high						';             
aWarningMessagesAsStrings[5] :=    	'RedLED No Supply Voltage							';                
aWarningMessagesAsStrings[6] :=    	'GreenLED Temperature too high						';           
aWarningMessagesAsStrings[7] :=    	'GreenLED No Supply Voltage							';              
aWarningMessagesAsStrings[8] :=    	'BlueLED Temperature too high						';            
aWarningMessagesAsStrings[9] :=    	'BlueLED No Supply Voltage							';               
aWarningMessagesAsStrings[10]:=     'EqualizingController Invalid Paramaters			';
aWarningMessagesAsStrings[11]:=     'EqualizingController Invalid CycleTime				'; 
aWarningMessagesAsStrings[12]:=     'TrajectoryGeneratorXMC1 AirGap OutOfRange			';                     
aWarningMessagesAsStrings[13]:=     'TrajectoryGeneratorXMC1 Velocity OutOfRange		';                    
aWarningMessagesAsStrings[14]:=     'TrajectoryGeneratorXMC1 Acceleration OutOfRange	';                 
aWarningMessagesAsStrings[15]:=     'TrajectoryGeneratorXMC1 Current OutOfRange			';                    
aWarningMessagesAsStrings[16]:=     'TrajectoryGeneratorXMC1 Voltage OutOfRange			';      
aWarningMessagesAsStrings[17]:=     'TrajectoryGeneratorXMC1 Force OutOfRange           ';
aWarningMessagesAsStrings[18]:=     'TrajectoryGeneratorXMC2 AirGap OutOfRange          ';
aWarningMessagesAsStrings[19]:=     'TrajectoryGeneratorXMC2 Velocity OutOfRange        ';
aWarningMessagesAsStrings[20]:=     'TrajectoryGeneratorXMC2 Acceleration OutOfRange    ';
aWarningMessagesAsStrings[21]:=     'TrajectoryGeneratorXMC2 Current OutOfRange         ';
aWarningMessagesAsStrings[22]:=     'TrajectoryGeneratorXMC2 Voltage OutOfRange         ';
aWarningMessagesAsStrings[23]:=     'TrajectoryGeneratorXMC2 Force OutOfRange           ';
aWarningMessagesAsStrings[24]:=     'TrajectoryGeneratorXMC3 AirGap OutOfRange          ';
aWarningMessagesAsStrings[25]:=     'TrajectoryGeneratorXMC3 Velocity OutOfRange        ';
aWarningMessagesAsStrings[26]:=     'TrajectoryGeneratorXMC3 Acceleration OutOfRange    ';
aWarningMessagesAsStrings[27]:=     'TrajectoryGeneratorXMC3 Current OutOfRange         ';
aWarningMessagesAsStrings[28]:=     'TrajectoryGeneratorXMC3 Voltage OutOfRange         ';
aWarningMessagesAsStrings[29]:=     'TrajectoryGeneratorXMC3 Force OutOfRange           ';
aWarningMessagesAsStrings[30]:=     'TrajectoryGeneratorXMC4 AirGap OutOfRange          ';
aWarningMessagesAsStrings[31]:=     'TrajectoryGeneratorXMC4 Velocity OutOfRange        ';
aWarningMessagesAsStrings[32]:=     'TrajectoryGeneratorXMC4 Acceleration OutOfRange    ';
aWarningMessagesAsStrings[33]:=     'TrajectoryGeneratorXMC4 Current OutOfRange         ';
aWarningMessagesAsStrings[34]:=     'TrajectoryGeneratorXMC4 Voltage OutOfRange         ';
aWarningMessagesAsStrings[35]:=     'TrajectoryGeneratorXMC4 Force OutOfRange	        ';  
aWarningMessagesAsStrings[36]:=     'IMU1 CommunicationError                            ';
aWarningMessagesAsStrings[37]:=     'IMU1 OutOfRange                                    ';
aWarningMessagesAsStrings[38]:=     'IMU2 CommunicationError                            ';
aWarningMessagesAsStrings[39]:=		'IMU2 OutOfRange                                    ';
aWarningMessagesAsStrings[40]:=		'GuidanceControllerXMC1 Current OutOfRange          ';
aWarningMessagesAsStrings[41]:=		'GuidanceControllerXMC1 Voltage OutOfRange          ';
aWarningMessagesAsStrings[42]:=		'GuidanceControllerXMC1 Force OutOfRange            ';
aWarningMessagesAsStrings[43]:=     'GuidanceControllerXMC2 Current OutOfRange          ';                     
aWarningMessagesAsStrings[44]:=     'GuidanceControllerXMC2 Voltage OutOfRange          ';
aWarningMessagesAsStrings[45]:=     'GuidanceControllerXMC2 Force OutOfRange            ';
aWarningMessagesAsStrings[46]:=     'GuidanceControllerXMC3 Current OutOfRange          ';
aWarningMessagesAsStrings[47]:=     'GuidanceControllerXMC3 Voltage OutOfRange          ';
aWarningMessagesAsStrings[48]:=     'GuidanceControllerXMC3 Force OutOfRange            ';
aWarningMessagesAsStrings[49]:=     'GuidanceControllerXMC4 Current OutOfRange          ';
aWarningMessagesAsStrings[50]:=     'GuidanceControllerXMC4 Voltage OutOfRange          ';
aWarningMessagesAsStrings[51]:=     'GuidanceControllerXMC4 Force OutOfRange            ';


FOR n := 0 TO PRG_ErrorHandling.nNumberOfWarnings-1 DO
	IF aWarningArray[n] THEN
		aCounterID[n] := aCounterID[n] + 1;
		IF aCounterID[n] = nCounterMax THEN
			aCounterID[n] := nCounterReset;
		END_IF
		fbEventMessage.CreateEx(stEventEntry:=TC_Events.MainControlEventClass.Warning, 0);
		IF aCounterID[n] = 1 THEN
			fbEventMessage.ipArguments.Clear().AddString(aWarningMessagesAsStrings[n]);
			fbEventMessage.Send(0);
		END_IF
	ELSE
		aCounterID[n] := 0;
	END_IF	
END_FOR


//ErrorMessages
//*Add New ErrorMessages here*
aErrorArray[0] := PRG_ErrorHandling.nErrorBits.0;
aErrorArray[1] := PRG_ErrorHandling.nErrorBits.1;
aErrorArray[2] := PRG_ErrorHandling.nErrorBits.2;
aErrorArray[3] := PRG_ErrorHandling.nErrorBits.3;
aErrorArray[4] := PRG_ErrorHandling.nErrorBits.4;
aErrorArray[5] := PRG_ErrorHandling.nErrorBits.5;

aErrorMessagesAsStrings[0] := 'Connection Timeout to Operation Control';
aErrorMessagesAsStrings[1] := 'Connection Timeout to XMC1';
aErrorMessagesAsStrings[2] := 'Connection Timeout to XMC2';
aErrorMessagesAsStrings[3] := 'Connection Timeout to XMC3';
aErrorMessagesAsStrings[4] := 'Connection Timeout to XMC4';
aErrorMessagesAsStrings[5] := 'EtherCAT Master Missing Ethernet Connection';

FOR n := 0 TO PRG_ErrorHandling.nNumberOfErrors - 1 DO
	IF aErrorArray[n] THEN
		aCounterID[n + PRG_ErrorHandling.nNumberOfWarnings] := aCounterID[n + PRG_ErrorHandling.nNumberOfWarnings] + 1;
		IF aCounterID[n + PRG_ErrorHandling.nNumberOfWarnings] = nCounterMax THEN
			aCounterID[n + PRG_ErrorHandling.nNumberOfWarnings] := nCounterReset;
		END_IF
		fbEventMessage.CreateEx(stEventEntry:=TC_Events.MainControlEventClass.Error, 0);
		IF aCounterID[n + PRG_ErrorHandling.nNumberOfWarnings] = 1 THEN
			fbEventMessage.ipArguments.Clear().AddString(sMainControllerStateAsString).AddString(aErrorMessagesAsStrings[n]);
			fbEventMessage.Send(0);
		END_IF
	ELSE
		aCounterID[n + PRG_ErrorHandling.nNumberOfWarnings] := 0;
	END_IF
END_FOR

PROPERTY PUBLIC aEventCounter : ARRAY [0..PRG_ErrorHandling.nNumberOfWarnings + PRG_ErrorHandling.nNumberOfErrors + PRG_ErrorHandling.nNumberOfInfos - 1] OF USINT
GET
VAR
	k : INT;
END_VAR
FOR k := 0 TO PRG_ErrorHandling.nNumberOfWarnings + PRG_ErrorHandling.nNumberOfErrors + PRG_ErrorHandling.nNumberOfInfos - 1 DO
	aEventCounter[k] := aCounterID[k];
END_FOR
END_GET
SET
VAR
	k : INT;
END_VAR
FOR k := 0 TO PRG_ErrorHandling.nNumberOfWarnings + PRG_ErrorHandling.nNumberOfErrors + PRG_ErrorHandling.nNumberOfInfos - 1 DO
	aCounterID[k] := aEventCounter[k];
END_FOR
END_SET
END_PROPERTY

END_FUNCTION_BLOCK

// ---- POUs/PRG_MainController.TcPOU
PROGRAM PRG_MainController
VAR
	fbServiceModule 			: FB_ServiceModule;
	fbLevitationSystem 			: FB_LevitationSystem;
	fbGuidanceSystem 			: FB_GuidanceSystem;
	
	eState 						: TopLevelSTM := TopLevelSTM.STARTUP;
	
	stOperationControlCommands 	: OperationControlCommands;
	stXMCCommands 				: XMCCommands;
END_VAR

doDataHandling();

CASE eState OF
	////
	TopLevelSTM.STARTUP:
		doEnableSystems();
		doCheckSystem();
		
		
		IF PRG_ErrorHandling.bStartUpCheck AND NOT PRG_ErrorHandling.bGoToError THEN
			eState := TopLevelSTM.READY;
		ELSE
			IF PRG_ErrorHandling.bErrorInStartUp OR PRG_ErrorHandling.bGoToError THEN
				fbServiceModule(eState:=ServiceModuleSTM.PreparingForError);
				eState := TopLevelSTM.ERROR;
			ELSE
				eState := TopLevelSTM.STARTUP;
			END_IF
		END_IF
	////
	TopLevelSTM.READY:
		fbServiceModule.eState := ServiceModuleSTM.Waiting;
		fbLevitationSystem.eState := LevitationSystemSTM.Stationary;
		fbGuidanceSystem.eState := GuidanceSystemSTM.PreRunning;
		stXMCCommands.bStopOperational := FALSE;
		stOperationControlCommands.bShutdownFinished := FALSE;
		
		fbServiceModule();
		fbLevitationSystem();
		fbGuidanceSystem();


		IF PRG_ErrorHandling.bErrorInReady OR PRG_ErrorHandling.bGoToError THEN
			fbServiceModule(eState := ServiceModuleSTM.PreparingForError);
			eState := TopLevelSTM.ERROR;
		ELSIF stOperationControlCommands.bStartOperational THEN
			stXMCCommands.bStartOperational := TRUE;	
			eState := TopLevelSTM.OPERATIONAL;
		END_IF
	////
	TopLevelSTM.OPERATIONAL:
		fbServiceModule.eState := ServiceModuleSTM.Running;
		stXMCCommands.bStartOperational := FALSE;
		
		IF fbLevitationSystem.bTrajectoryCompleted THEN
			fbLevitationSystem.eState := LevitationSystemSTM.HoldingAirGap;
		ELSE
			fbLevitationSystem.eState := LevitationSystemSTM.Transitioning;
		END_IF
		
		IF stOperationControlCommands.bMinimumAirGapForGC THEN
			fbGuidanceSystem.eState := GuidanceSystemSTM.Running;
		ELSE
			fbGuidanceSystem.eState := GuidanceSystemSTM.PreRunning;
		END_IF
		
		fbServiceModule();
		fbLevitationSystem();
		fbGuidanceSystem();
		
		
		IF PRG_ErrorHandling.bErrorInOperational OR PRG_ErrorHandling.bGoToError OR stOperationControlCommands.bStopOperational THEN
			eState := TopLevelSTM.SHUTDOWN;
		END_IF
	////
	TopLevelSTM.SHUTDOWN:
		fbServiceModule.eState := ServiceModuleSTM.PostRunning;
		
		fbLevitationSystem.eState := LevitationSystemSTM.TransitioningToZero;
		
		IF stOperationControlCommands.bMinimumAirGapForGC THEN
			fbGuidanceSystem.eState := GuidanceSystemSTM.Running;
		ELSE
			fbGuidanceSystem.eState := GuidanceSystemSTM.PostRunning;
		END_IF
		
		fbServiceModule();
		fbLevitationSystem();
		fbGuidanceSystem();
		
		IF fbLevitationSystem.bTrajectoryCompleted OR PRG_ErrorHandling.fbShutdownTimer.Q THEN
			stOperationControlCommands.bShutdownFinished := TRUE;
			
			IF PRG_ErrorHandling.bErrorInOperational OR PRG_ErrorHandling.bErrorInShutdown OR PRG_ErrorHandling.bGoToError THEN
				fbServiceModule(eState := ServiceModuleSTM.PreparingForError);
				eState := TopLevelSTM.ERROR;
			ELSIF stOperationControlCommands.bEndShutdown THEN
				stXMCCommands.bStopOperational := TRUE;
				eState := TopLevelSTM.READY;
			END_IF
		END_IF
		

	////	
	TopLevelSTM.ERROR:
		IF PRG_ErrorHandling.bAllErrorsAcknowledged THEN
			stXMCCommands.bAckError := TRUE;
			eState := TopLevelSTM.STARTUP;
		END_IF
END_CASE

METHOD PRIVATE doCheckSystem
VAR_INPUT
END_VAR
fbServiceModule(eState := ServiceModuleSTM.Idling);
fbLevitationSystem(eState := LevitationSystemSTM.Idling);
fbGuidanceSystem(eState := GuidanceSystemSTM.Idling);

stXMCCommands.bAckError := FALSE;
stXMCCommands.bStartOperational := FALSE;
stXMCCommands.bStopOperational := FALSE;
END_METHOD

METHOD PRIVATE doDataHandling
VAR_INPUT
END_VAR
VAR
	aTempArray0 : ARRAY [0..2] OF REAL;
	aTempArray1 : ARRAY [0..2] OF REAL;
	aTempArray2 : ARRAY [0..3] OF REAL;
	aTempArray3 : ARRAY [0..3] OF REAL;
	aTempArray4 : ARRAY [0..3] OF REAL;
	aTempArray5 : ARRAY [0..3] OF REAL;
	aTempArray6 : ARRAY [0..3] OF REAL;
	aTempArray7 : ARRAY [0..3] OF REAL;
	aTempArray8 : ARRAY [0..3] OF REAL;
	aTempArray9 : ARRAY [0..3] OF REAL;
	aTempArray10 : ARRAY [0..3] OF REAL;
	aTempArray11 : ARRAY [0..3] OF REAL;
	aTempArray12 : ARRAY [0..3] OF REAL;
	aTempArray13 : ARRAY [0..3] OF REAL;
	aTempArray14 : ARRAY [0..3] OF REAL;
	aTempArray15 : ARRAY [0..3] OF REAL;
	aTempArray16 : ARRAY [0..3] OF REAL;
	aTempArray17 : ARRAY [0..3] OF REAL;
	aTempArray18 : ARRAY [0..3] OF REAL;
	aTempArray19 : ARRAY [0..3] OF REAL;
END_VAR
//ArrayHandling
aTempArray0 := PRG_MainController.fbGuidanceSystem.aIMU1Acceleration;
aTempArray1 := PRG_MainController.fbGuidanceSystem.aIMU2Acceleration;
aTempArray2 := PRG_MainController.fbLevitationSystem.aECOutputZVector;
aTempArray3 := PRG_MainController.fbLevitationSystem.aTGOutputLevDistance;
aTempArray4 := PRG_MainController.fbLevitationSystem.aTGOutputLevVelocity;
aTempArray5 := PRG_MainController.fbLevitationSystem.aTGOutputLevAcceleration;
aTempArray6 := PRG_MainController.fbLevitationSystem.aTGOutputLevCurrent;
aTempArray7 := PRG_MainController.fbLevitationSystem.aTGOutputLevVoltage;
aTempArray8 := PRG_MainController.fbLevitationSystem.aTGOutputLevForce;
aTempArray9 := PRG_MainController.fbGuidanceSystem.aGCOutputGuidCurrent;
aTempArray10 := PRG_MainController.fbGuidanceSystem.aGCOutputGuidVoltage;
aTempArray11 := PRG_MainController.fbGuidanceSystem.aGCOutputGuidForce;

PRG_MainController.fbLevitationSystem.aTGActualLevDistance				:=		aTempArray12;
PRG_MainController.fbLevitationSystem.aTGActualLevVelocity              :=      aTempArray13;
PRG_MainController.fbLevitationSystem.aTGActualLevAcceleration          :=      aTempArray14;
PRG_MainController.fbLevitationSystem.aTGActualLevCurrent               :=      aTempArray15;
PRG_MainController.fbGuidanceSystem.aGCActualGuidDistance               :=      aTempArray16;
PRG_MainController.fbGuidanceSystem.aGCActualGuidAcceleration           :=      aTempArray17;                                                             
PRG_MainController.fbGuidanceSystem.aGCActualGuidCurrent			    :=      aTempArray18;   





//OperationControlData
	//From OC to MC
		//Main Controller
		PRG_MainController.stOperationControlCommands.bStartOperational			:= 			OperationControlData.stFromOCToMC.OM_origO_StartOperational;     
		PRG_MainController.stOperationControlCommands.bStopOperational			:= 			OperationControlData.stFromOCToMC.OM_origO_StopOperational;		
		PRG_MainController.stOperationControlCommands.bEndShutdown				:= 			OperationControlData.stFromOCToMC.OM_origO_EndShutdown;			
		PRG_MainController.stOperationControlCommands.bGoToError				:= 			OperationControlData.stFromOCToMC.OM_origO_GoToError;              
		PRG_MainController.stOperationControlCommands.bAckError					:= 			OperationControlData.stFromOCToMC.OM_origO_AckError;				
		PRG_MainController.stOperationControlCommands.nOperationMode.0			:= 			OperationControlData.stFromOCToMC.OM_origG_ServiceModuleDisable;	
		PRG_MainController.stOperationControlCommands.nOperationMode.1			:= 			OperationControlData.stFromOCToMC.OM_origG_LevitationDisable;      
		PRG_MainController.stOperationControlCommands.nOperationMode.2			:= 			OperationControlData.stFromOCToMC.OM_origG_GuidanceDisable;        
		PRG_MainController.stOperationControlCommands.nSafetyCounterOC			:= 			OperationControlData.stFromOCToMC.OM_origO_SafetyCounter;          											
		//Levitation
		PRG_MainController.fbLevitationSystem.nTGControlOption					:= 			OperationControlData.stFromOCToMC.OM_origG_LevControlOption;		
		PRG_MainController.fbLevitationSystem.fTGDesiredLevDistance				:= 			OperationControlData.stFromOCToMC.OM_origG_DesiredLevDistance;		
		PRG_MainController.fbLevitationSystem.fTGDesiredLevVelocity				:= 			OperationControlData.stFromOCToMC.OM_origG_DesiredLevVelocity;		
		PRG_MainController.fbLevitationSystem.fTGDesiredLevAcceleration			:= 			OperationControlData.stFromOCToMC.OM_origG_DesiredLevAcceleration;	
		PRG_MainController.fbLevitationSystem.fTGDesiredLevTime					:= 			OperationControlData.stFromOCToMC.OM_origG_DesiredLevTime;									
		//Guidance
		PRG_MainController.stOperationControlCommands.bMinimumAirGapForGC		:= 			OperationControlData.stFromOCToMC.OM_origG_EnableGuidController;	
		PRG_MainController.fbGuidanceSystem.aGCReferenceYSignal					:= 			OperationControlData.stFromOCToMC.OM_origG_GuidReferenceYSignal;
		PRG_MainController.fbGuidanceSystem.nGCControlOption					:= 			OperationControlData.stFromOCToMC.OM_origG_GuidControlOption;			

	//From MC to OC
		//Main Controller
		OperationControlData.stFromMCToOC.MO_origM_State						:=			PRG_MainController.eState;
		OperationControlData.stFromMCToOC.MO_origM_WarnBits						:=			PRG_ErrorHandling.nWarningBits;
		OperationControlData.stFromMCToOC.MO_origM_ErrBits						:=			PRG_ErrorHandling.nErrorBits;
		OperationControlData.stFromMCToOC.MO_origM_SafetyCounter				:=			PRG_ErrorHandling.fbSafetyCounter.nSafetyCounter;
		OperationControlData.stFromMCToOC.MO_origM_ShutdownFinished				:=			PRG_MainController.stOperationControlCommands.bShutdownFinished;
		//ServiceModule
		OperationControlData.stFromMCToOC.MO_origM_DistanceServiceModule		:=			PRG_MainController.fbServiceModule.fDistance;
		//Levitation
		OperationControlData.stFromMCToOC.MO_origM_ECOutputDistanceXMC1			:=			aTempArray2[0];
		OperationControlData.stFromMCToOC.MO_origM_ECOutputDistanceXMC2			:=			aTempArray2[1];
		OperationControlData.stFromMCToOC.MO_origM_ECOutputDistanceXMC3			:=			aTempArray2[2];
		OperationControlData.stFromMCToOC.MO_origM_ECOutputDistanceXMC4			:=			aTempArray2[3];
		OperationControlData.stFromMCToOC.MO_origM_TGOutputLevDistanceXMC1		:=			aTempArray3[0];
		OperationControlData.stFromMCToOC.MO_origM_TGOutputLevDistanceXMC2		:=			aTempArray3[1];
		OperationControlData.stFromMCToOC.MO_origM_TGOutputLevDistanceXMC3		:=			aTempArray3[2];
		OperationControlData.stFromMCToOC.MO_origM_TGOutputLevDistanceXMC4		:=			aTempArray3[3];
		OperationControlData.stFromMCToOC.MO_origM_TGOutputLevVelocityXMC1		:=			aTempArray4[0];
		OperationControlData.stFromMCToOC.MO_origM_TGOutputLevVelocityXMC2		:=			aTempArray4[1];
		OperationControlData.stFromMCToOC.MO_origM_TGOutputLevVelocityXMC3		:=			aTempArray4[2];
		OperationControlData.stFromMCToOC.MO_origM_TGOutputLevVelocityXMC4		:=			aTempArray4[3];
		OperationControlData.stFromMCToOC.MO_origM_TGOutputLevAccelerationXMC1	:=			aTempArray5[0];
		OperationControlData.stFromMCToOC.MO_origM_TGOutputLevAccelerationXMC2	:=			aTempArray5[1];
		OperationControlData.stFromMCToOC.MO_origM_TGOutputLevAccelerationXMC3	:=			aTempArray5[2];
		OperationControlData.stFromMCToOC.MO_origM_TGOutputLevAccelerationXMC4	:=			aTempArray5[3];
		OperationControlData.stFromMCToOC.MO_origM_TGOutputLevCurrentXMC1		:=			aTempArray6[0];
		OperationControlData.stFromMCToOC.MO_origM_TGOutputLevCurrentXMC2		:=			aTempArray6[1];
		OperationControlData.stFromMCToOC.MO_origM_TGOutputLevCurrentXMC3		:=			aTempArray6[2];
		OperationControlData.stFromMCToOC.MO_origM_TGOutputLevCurrentXMC4		:=			aTempArray6[3];
		OperationControlData.stFromMCToOC.MO_origM_TGOutputLevVoltageXMC1		:=			aTempArray7[0];
		OperationControlData.stFromMCToOC.MO_origM_TGOutputLevVoltageXMC2		:=			aTempArray7[1];
		OperationControlData.stFromMCToOC.MO_origM_TGOutputLevVoltageXMC3		:=			aTempArray7[2];
		OperationControlData.stFromMCToOC.MO_origM_TGOutputLevVoltageXMC4		:=			aTempArray7[3];
		OperationControlData.stFromMCToOC.MO_origM_TGOutputLevForceXMC1			:=			aTempArray8[0];
		OperationControlData.stFromMCToOC.MO_origM_TGOutputLevForceXMC2			:=			aTempArray8[1];
		OperationControlData.stFromMCToOC.MO_origM_TGOutputLevForceXMC3			:=			aTempArray8[2];
		OperationControlData.stFromMCToOC.MO_origM_TGOutputLevForceXMC4			:=			aTempArray8[3];
		//Guidance
		OperationControlData.stFromMCToOC.MO_origM_GuidanceIMUX0				:=			aTempArray0[0];
		OperationControlData.stFromMCToOC.MO_origM_GuidanceIMUY0				:=			aTempArray0[1];
		OperationControlData.stFromMCToOC.MO_origM_GuidanceIMUZ0				:=			aTempArray0[2];
		OperationControlData.stFromMCToOC.MO_origM_GuidanceIMUX1				:=			aTempArray1[0];
		OperationControlData.stFromMCToOC.MO_origM_GuidanceIMUY1				:=			aTempArray1[1];
		OperationControlData.stFromMCToOC.MO_origM_GuidanceIMUZ1				:=			aTempArray1[2];
		OperationControlData.stFromMCToOC.MO_origM_GCOutputGuidCurrentXMC1		:=			aTempArray9[0];
		OperationControlData.stFromMCToOC.MO_origM_GCOutputGuidCurrentXMC2		:=			aTempArray9[1];
		OperationControlData.stFromMCToOC.MO_origM_GCOutputGuidCurrentXMC3		:=			aTempArray9[2];
		OperationControlData.stFromMCToOC.MO_origM_GCOutputGuidCurrentXMC4		:=			aTempArray9[3];
		OperationControlData.stFromMCToOC.MO_origM_GCOutputGuidVoltageXMC1		:=			aTempArray10[0];
		OperationControlData.stFromMCToOC.MO_origM_GCOutputGuidVoltageXMC2		:=			aTempArray10[1];
		OperationControlData.stFromMCToOC.MO_origM_GCOutputGuidVoltageXMC3		:=			aTempArray10[2];
		OperationControlData.stFromMCToOC.MO_origM_GCOutputGuidVoltageXMC4		:=			aTempArray10[3];
		OperationControlData.stFromMCToOC.MO_origM_GCOutputGuidForceXMC1		:=			aTempArray11[0];
		OperationControlData.stFromMCToOC.MO_origM_GCOutputGuidForceXMC2		:=			aTempArray11[1];
		OperationControlData.stFromMCToOC.MO_origM_GCOutputGuidForceXMC3		:=			aTempArray11[2];
		OperationControlData.stFromMCToOC.MO_origM_GCOutputGuidForceXMC4		:=			aTempArray11[3];



//XMC Data
	//From XMC to MC
		//Sensor Values
		aTempArray12[0]															:=			XMCData.stFromXMC1ToMC.EM_origE_DistanceLevitationFiltered;					
		aTempArray12[1]															:=			XMCData.stFromXMC2ToMC.EM_origE_DistanceLevitationFiltered	;				
		aTempArray12[2]															:=			XMCData.stFromXMC3ToMC.EM_origE_DistanceLevitationFiltered	;				
		aTempArray12[3]															:=			XMCData.stFromXMC4ToMC.EM_origE_DistanceLevitationFiltered	;		
		aTempArray13[0]															:=			XMCData.stFromXMC1ToMC.EM_origE_VelocityZFiltered	;				
		aTempArray13[1]															:=			XMCData.stFromXMC2ToMC.EM_origE_VelocityZFiltered	;				
		aTempArray13[2]															:=			XMCData.stFromXMC3ToMC.EM_origE_VelocityZFiltered	;				
		aTempArray13[3]															:=			XMCData.stFromXMC4ToMC.EM_origE_VelocityZFiltered	;	
		aTempArray14[0]															:=			XMCData.stFromXMC1ToMC.EM_origE_IMUZ				;			
		aTempArray14[1]															:=			XMCData.stFromXMC2ToMC.EM_origE_IMUZ				;			
		aTempArray14[2]															:=			XMCData.stFromXMC3ToMC.EM_origE_IMUZ				;			
		aTempArray14[3]															:=			XMCData.stFromXMC4ToMC.EM_origE_IMUZ				;	
		aTempArray15[0]															:=			DINT_TO_REAL(XMCData.stFromXMC1ToMC.EM_origE_CurrentLev)			;				
		aTempArray15[1]															:=			DINT_TO_REAL(XMCData.stFromXMC2ToMC.EM_origE_CurrentLev)			;				
		aTempArray15[2]															:=			DINT_TO_REAL(XMCData.stFromXMC3ToMC.EM_origE_CurrentLev	)		;				
		aTempArray15[3]															:=			DINT_TO_REAL(XMCData.stFromXMC4ToMC.EM_origE_CurrentLev	)		;		
		aTempArray16[0]															:=			XMCData.stFromXMC1ToMC.EM_origE_DistanceGuidanceFiltered;				
		aTempArray16[1]															:=			XMCData.stFromXMC2ToMC.EM_origE_DistanceGuidanceFiltered;				
		aTempArray16[2]															:=			XMCData.stFromXMC3ToMC.EM_origE_DistanceGuidanceFiltered;				
		aTempArray16[3]															:=			XMCData.stFromXMC4ToMC.EM_origE_DistanceGuidanceFiltered;		
		aTempArray17[0]															:=			XMCData.stFromXMC1ToMC.EM_origE_IMUY				;			
		aTempArray17[1]															:=			XMCData.stFromXMC2ToMC.EM_origE_IMUY				;			
		aTempArray17[2]															:=			XMCData.stFromXMC3ToMC.EM_origE_IMUY				;			
		aTempArray17[3]															:=			XMCData.stFromXMC4ToMC.EM_origE_IMUY				;	
		aTempArray18[0]															:=			DINT_TO_REAL(XMCData.stFromXMC1ToMC.EM_origE_CurrentGuid)			;				
		aTempArray18[1]															:=			DINT_TO_REAL(XMCData.stFromXMC2ToMC.EM_origE_CurrentGuid)			;				
		aTempArray18[2]															:=			DINT_TO_REAL(XMCData.stFromXMC3ToMC.EM_origE_CurrentGuid)			;				
		aTempArray18[3]															:=			DINT_TO_REAL(XMCData.stFromXMC4ToMC.EM_origE_CurrentGuid)			;	
		//System Status
		PRG_MainController.stXMCCommands.nSafetyCounterXMC1						:=			XMCData.stFromXMC1ToMC.EM_origE_SafetyCounter		;					 			
		PRG_MainController.stXMCCommands.nSafetyCounterXMC2						:=			XMCData.stFromXMC2ToMC.EM_origE_SafetyCounter		;					 			
		PRG_MainController.stXMCCommands.nSafetyCounterXMC3						:=			XMCData.stFromXMC3ToMC.EM_origE_SafetyCounter		;					 			
		PRG_MainController.stXMCCommands.nSafetyCounterXMC4			        	:=			XMCData.stFromXMC4ToMC.EM_origE_SafetyCounter	;
		PRG_MainController.stXMCCommands.nStateXMC1								:=			XMCData.stFromXMC1ToMC.EM_origE_State;
		PRG_MainController.stXMCCommands.nStateXMC2								:=			XMCData.stFromXMC2ToMC.EM_origE_State;
		PRG_MainController.stXMCCommands.nStateXMC3								:=			XMCData.stFromXMC3ToMC.EM_origE_State;
		PRG_MainController.stXMCCommands.nStateXMC4								:=			XMCData.stFromXMC4ToMC.EM_origE_State;
		
	//From MC to XMC
		//Control
		XMCData.stFromMCToXMC1.ME_origM_SafetyCounter							:=			PRG_ErrorHandling.fbSafetyCounter.nSafetyCounter;
		XMCData.stFromMCToXMC2.ME_origM_SafetyCounter							:=			PRG_ErrorHandling.fbSafetyCounter.nSafetyCounter;
		XMCData.stFromMCToXMC3.ME_origM_SafetyCounter							:=			PRG_ErrorHandling.fbSafetyCounter.nSafetyCounter;
		XMCData.stFromMCToXMC4.ME_origM_SafetyCounter							:=			PRG_ErrorHandling.fbSafetyCounter.nSafetyCounter;		
		XMCData.stFromMCToXMC1.ME_origM_StartOperational						:=			PRG_MainController.stXMCCommands.bStartOperational;
		XMCData.stFromMCToXMC2.ME_origM_StartOperational						:=			PRG_MainController.stXMCCommands.bStartOperational;
		XMCData.stFromMCToXMC3.ME_origM_StartOperational						:=			PRG_MainController.stXMCCommands.bStartOperational;
		XMCData.stFromMCToXMC4.ME_origM_StartOperational						:=			PRG_MainController.stXMCCommands.bStartOperational;		
		XMCData.stFromMCToXMC1.ME_origM_StopOperational							:=			PRG_MainController.stXMCCommands.bStopOperational;
		XMCData.stFromMCToXMC2.ME_origM_StopOperational							:=			PRG_MainController.stXMCCommands.bStopOperational;
		XMCData.stFromMCToXMC3.ME_origM_StopOperational							:=			PRG_MainController.stXMCCommands.bStopOperational;
		XMCData.stFromMCToXMC4.ME_origM_StopOperational							:=			PRG_MainController.stXMCCommands.bStopOperational;			
		XMCData.stFromMCToXMC1.ME_origM_AckError								:=			PRG_MainController.stXMCCommands.bAckError;
		XMCData.stFromMCToXMC2.ME_origM_AckError								:=			PRG_MainController.stXMCCommands.bAckError;
		XMCData.stFromMCToXMC3.ME_origM_AckError								:=			PRG_MainController.stXMCCommands.bAckError;
		XMCData.stFromMCToXMC4.ME_origM_AckError								:=			PRG_MainController.stXMCCommands.bAckError;	
		XMCData.stFromMCToXMC1.ME_origM_DebugSel								:=			PRG_MainController.stXMCCommands.nDebugPWMSel;
		XMCData.stFromMCToXMC2.ME_origM_DebugSel								:=			PRG_MainController.stXMCCommands.nDebugPWMSel;
		XMCData.stFromMCToXMC3.ME_origM_DebugSel								:=			PRG_MainController.stXMCCommands.nDebugPWMSel;
		XMCData.stFromMCToXMC4.ME_origM_DebugSel								:=			PRG_MainController.stXMCCommands.nDebugPWMSel;			
		XMCData.stFromMCToXMC1.ME_origM_DebugPWMLev								:=			PRG_MainController.stXMCCommands.nDebugPWMLev;
		XMCData.stFromMCToXMC2.ME_origM_DebugPWMLev								:=			PRG_MainController.stXMCCommands.nDebugPWMLev;
		XMCData.stFromMCToXMC3.ME_origM_DebugPWMLev								:=			PRG_MainController.stXMCCommands.nDebugPWMLev;
		XMCData.stFromMCToXMC4.ME_origM_DebugPWMLev								:=			PRG_MainController.stXMCCommands.nDebugPWMLev;		
		XMCData.stFromMCToXMC1.ME_origM_DebugPWMGuid							:=			PRG_MainController.stXMCCommands.nDebugPWMGuid;
		XMCData.stFromMCToXMC2.ME_origM_DebugPWMGuid							:=			PRG_MainController.stXMCCommands.nDebugPWMGuid;
		XMCData.stFromMCToXMC3.ME_origM_DebugPWMGuid							:=			PRG_MainController.stXMCCommands.nDebugPWMGuid;
		XMCData.stFromMCToXMC4.ME_origM_DebugPWMGuid							:=			PRG_MainController.stXMCCommands.nDebugPWMGuid;			
		//Guidance
		XMCData.stFromMCToXMC1.ME_origM_DesiredGuidCurrent					:=			aTempArray9[0];
		XMCData.stFromMCToXMC2.ME_origM_DesiredGuidCurrent					:=			aTempArray9[1];
		XMCData.stFromMCToXMC3.ME_origM_DesiredGuidCurrent					:=			aTempArray9[2];
		XMCData.stFromMCToXMC4.ME_origM_DesiredGuidCurrent					:=			aTempArray9[3];		
		XMCData.stFromMCToXMC1.ME_origM_DesiredGuidForce					:=			aTempArray11[0];
		XMCData.stFromMCToXMC2.ME_origM_DesiredGuidForce					:=			aTempArray11[1];
		XMCData.stFromMCToXMC3.ME_origM_DesiredGuidForce					:=			aTempArray11[2];
		XMCData.stFromMCToXMC4.ME_origM_DesiredGuidForce					:=			aTempArray11[3];
		XMCData.stFromMCToXMC1.ME_origM_DesiredGuidVoltage					:=			aTempArray10[0];
		XMCData.stFromMCToXMC2.ME_origM_DesiredGuidVoltage					:=			aTempArray10[1];
		XMCData.stFromMCToXMC3.ME_origM_DesiredGuidVoltage					:=			aTempArray10[2];
		XMCData.stFromMCToXMC4.ME_origM_DesiredGuidVoltage					:=			aTempArray10[3];		
		XMCData.stFromMCToXMC1.ME_origM_GuidEnableCurrentController				:=			PRG_MainController.fbGuidanceSystem.bEnableCurrentController;
		XMCData.stFromMCToXMC2.ME_origM_GuidEnableCurrentController				:=			PRG_MainController.fbGuidanceSystem.bEnableCurrentController;
		XMCData.stFromMCToXMC3.ME_origM_GuidEnableCurrentController				:=			PRG_MainController.fbGuidanceSystem.bEnableCurrentController;
		XMCData.stFromMCToXMC4.ME_origM_GuidEnableCurrentController				:=			PRG_MainController.fbGuidanceSystem.bEnableCurrentController;		
		XMCData.stFromMCToXMC1.ME_origM_GuidEnableIControl						:=			PRG_MainController.fbGuidanceSystem.bEnableIControl;
		XMCData.stFromMCToXMC2.ME_origM_GuidEnableIControl						:=			PRG_MainController.fbGuidanceSystem.bEnableIControl;
		XMCData.stFromMCToXMC3.ME_origM_GuidEnableIControl						:=			PRG_MainController.fbGuidanceSystem.bEnableIControl;
		XMCData.stFromMCToXMC4.ME_origM_GuidEnableIControl						:=			PRG_MainController.fbGuidanceSystem.bEnableIControl;		
		XMCData.stFromMCToXMC1.ME_origM_GuidEnablePControl						:=			PRG_MainController.fbGuidanceSystem.bEnableIControl;
		XMCData.stFromMCToXMC2.ME_origM_GuidEnablePControl						:=			PRG_MainController.fbGuidanceSystem.bEnableIControl;
		XMCData.stFromMCToXMC3.ME_origM_GuidEnablePControl						:=			PRG_MainController.fbGuidanceSystem.bEnableIControl;
		XMCData.stFromMCToXMC4.ME_origM_GuidEnablePControl						:=			PRG_MainController.fbGuidanceSystem.bEnableIControl;			
		//Levitation
		XMCData.stFromMCToXMC1.ME_origM_DesiredLevDistance					:=			aTempArray3[0] + aTempArray2[0];
		XMCData.stFromMCToXMC2.ME_origM_DesiredLevDistance					:=			aTempArray3[1] + aTempArray2[1];
		XMCData.stFromMCToXMC3.ME_origM_DesiredLevDistance					:=			aTempArray3[2] + aTempArray2[2];
		XMCData.stFromMCToXMC4.ME_origM_DesiredLevDistance					:=			aTempArray3[3] + aTempArray2[3];		
		XMCData.stFromMCToXMC1.ME_origM_DesiredLevVelocity					:=			aTempArray4[0];
		XMCData.stFromMCToXMC2.ME_origM_DesiredLevVelocity					:=			aTempArray4[1];
		XMCData.stFromMCToXMC3.ME_origM_DesiredLevVelocity					:=			aTempArray4[2];
		XMCData.stFromMCToXMC4.ME_origM_DesiredLevVelocity					:=			aTempArray4[3];		
		XMCData.stFromMCToXMC1.ME_origM_DesiredLevAcceleration				:=			aTempArray5[0];
		XMCData.stFromMCToXMC2.ME_origM_DesiredLevAcceleration				:=			aTempArray5[1];
		XMCData.stFromMCToXMC3.ME_origM_DesiredLevAcceleration				:=			aTempArray5[2];
		XMCData.stFromMCToXMC4.ME_origM_DesiredLevAcceleration				:=			aTempArray5[3];			
		XMCData.stFromMCToXMC1.ME_origM_DesiredLevCurrent					:=			aTempArray6[0];
		XMCData.stFromMCToXMC2.ME_origM_DesiredLevCurrent					:=			aTempArray6[1];
		XMCData.stFromMCToXMC3.ME_origM_DesiredLevCurrent					:=			aTempArray6[2];
		XMCData.stFromMCToXMC4.ME_origM_DesiredLevCurrent					:=			aTempArray6[3];	
		XMCData.stFromMCToXMC1.ME_origM_DesiredLevVoltage					:=			aTempArray7[0];
		XMCData.stFromMCToXMC2.ME_origM_DesiredLevVoltage					:=			aTempArray7[1];
		XMCData.stFromMCToXMC3.ME_origM_DesiredLevVoltage					:=			aTempArray7[2];
		XMCData.stFromMCToXMC4.ME_origM_DesiredLevVoltage					:=			aTempArray7[3];		
		XMCData.stFromMCToXMC1.ME_origM_DesiredLevForce					:=			aTempArray8[0];
		XMCData.stFromMCToXMC2.ME_origM_DesiredLevForce					:=			aTempArray8[1];
		XMCData.stFromMCToXMC3.ME_origM_DesiredLevForce					:=			aTempArray8[2];
		XMCData.stFromMCToXMC4.ME_origM_DesiredLevForce					:=			aTempArray8[3];		
		XMCData.stFromMCToXMC1.ME_origM_LevEnableCurrentController				:=			PRG_MainController.fbLevitationSystem.bEnableCurrentController;
		XMCData.stFromMCToXMC2.ME_origM_LevEnableCurrentController				:=			PRG_MainController.fbLevitationSystem.bEnableCurrentController;
		XMCData.stFromMCToXMC3.ME_origM_LevEnableCurrentController				:=			PRG_MainController.fbLevitationSystem.bEnableCurrentController;
		XMCData.stFromMCToXMC4.ME_origM_LevEnableCurrentController				:=			PRG_MainController.fbLevitationSystem.bEnableCurrentController;
		XMCData.stFromMCToXMC1.ME_origM_LevEnableIControl						:=			PRG_MainController.fbLevitationSystem.bEnableIControl;
		XMCData.stFromMCToXMC2.ME_origM_LevEnableIControl						:=			PRG_MainController.fbLevitationSystem.bEnableIControl;
		XMCData.stFromMCToXMC3.ME_origM_LevEnableIControl						:=			PRG_MainController.fbLevitationSystem.bEnableIControl;
		XMCData.stFromMCToXMC4.ME_origM_LevEnableIControl						:=			PRG_MainController.fbLevitationSystem.bEnableIControl;
		XMCData.stFromMCToXMC1.ME_origM_LevEnablePControl						:=			PRG_MainController.fbLevitationSystem.bEnableIControl;
		XMCData.stFromMCToXMC2.ME_origM_LevEnablePControl						:=			PRG_MainController.fbLevitationSystem.bEnableIControl;
		XMCData.stFromMCToXMC3.ME_origM_LevEnablePControl						:=			PRG_MainController.fbLevitationSystem.bEnableIControl;
		XMCData.stFromMCToXMC4.ME_origM_LevEnablePControl						:=			PRG_MainController.fbLevitationSystem.bEnableIControl;
		//Forward from GUI
		XMCData.stFromMCToXMC1.ME_origG_GuidControlOption						:=			OperationControlData.stFromOCToMC.OM_origG_GuidControlOption;
		XMCData.stFromMCToXMC2.ME_origG_GuidControlOption						:=			OperationControlData.stFromOCToMC.OM_origG_GuidControlOption;
		XMCData.stFromMCToXMC3.ME_origG_GuidControlOption						:=			OperationControlData.stFromOCToMC.OM_origG_GuidControlOption;
		XMCData.stFromMCToXMC4.ME_origG_GuidControlOption						:=			OperationControlData.stFromOCToMC.OM_origG_GuidControlOption;
		XMCData.stFromMCToXMC1.ME_origG_LevControlOption						:=			OperationControlData.stFromOCToMC.OM_origG_LevControlOption;
		XMCData.stFromMCToXMC2.ME_origG_LevControlOption						:=			OperationControlData.stFromOCToMC.OM_origG_LevControlOption;
		XMCData.stFromMCToXMC3.ME_origG_LevControlOption						:=			OperationControlData.stFromOCToMC.OM_origG_LevControlOption;
		XMCData.stFromMCToXMC4.ME_origG_LevControlOption						:=			OperationControlData.stFromOCToMC.OM_origG_LevControlOption;
		XMCData.stFromMCToXMC1.ME_origG_EnableGuidController					:=			OperationControlData.stFromOCToMC.OM_origG_EnableGuidController;
		XMCData.stFromMCToXMC2.ME_origG_EnableGuidController					:=			OperationControlData.stFromOCToMC.OM_origG_EnableGuidController;
		XMCData.stFromMCToXMC3.ME_origG_EnableGuidController					:=			OperationControlData.stFromOCToMC.OM_origG_EnableGuidController;
		XMCData.stFromMCToXMC4.ME_origG_EnableGuidController					:=			OperationControlData.stFromOCToMC.OM_origG_EnableGuidController;
		XMCData.stFromMCToXMC1.ME_origG_Logging_CounterOut						:=			OperationControlData.stFromOCToMC.OM_origG_LoggingCounterOut;
		XMCData.stFromMCToXMC2.ME_origG_Logging_CounterOut						:=			OperationControlData.stFromOCToMC.OM_origG_LoggingCounterOut;
		XMCData.stFromMCToXMC3.ME_origG_Logging_CounterOut						:=			OperationControlData.stFromOCToMC.OM_origG_LoggingCounterOut;
		XMCData.stFromMCToXMC4.ME_origG_Logging_CounterOut						:=			OperationControlData.stFromOCToMC.OM_origG_LoggingCounterOut;

//Forward XMC to OC
	//XMC1
		OperationControlData.stForwardXMC1ToOC.MO_origE_CurrentGuid				:=			XMCData.stFromXMC1ToMC.EM_origE_CurrentGuid;			
		OperationControlData.stForwardXMC1ToOC.MO_origE_CurrentLev				:=			XMCData.stFromXMC1ToMC.EM_origE_CurrentLev;		
		OperationControlData.stForwardXMC1ToOC.MO_origE_DistanceRawLev11		:=			XMCData.stFromXMC1ToMC.EM_origE_DistanceRawLev11;		
		OperationControlData.stForwardXMC1ToOC.MO_origE_DistanceRawLev12		:=			XMCData.stFromXMC1ToMC.EM_origE_DistanceRawLev12;		
		OperationControlData.stForwardXMC1ToOC.MO_origE_DistanceRawLev21		:=			XMCData.stFromXMC1ToMC.EM_origE_DistanceRawLev21;		
		OperationControlData.stForwardXMC1ToOC.MO_origE_DistanceRawLev22		:=			XMCData.stFromXMC1ToMC.EM_origE_DistanceRawLev22;		
		OperationControlData.stForwardXMC1ToOC.MO_origE_DistanceRawGuid11		:=			XMCData.stFromXMC1ToMC.EM_origE_DistanceRawGuid11;		
		OperationControlData.stForwardXMC1ToOC.MO_origE_DistanceRawGuid12		:=			XMCData.stFromXMC1ToMC.EM_origE_DistanceRawGuid12;		
		OperationControlData.stForwardXMC1ToOC.MO_origE_DistanceGuidanceFiltered	:=			XMCData.stFromXMC1ToMC.EM_origE_DistanceGuidanceFiltered;		
		OperationControlData.stForwardXMC1ToOC.MO_origE_DistanceLevitationFiltered		:=			XMCData.stFromXMC1ToMC.EM_origE_DistanceLevitationFiltered;	
		OperationControlData.stForwardXMC1ToOC.MO_origE_VelocityZFiltered		:=			XMCData.stFromXMC1ToMC.EM_origE_VelocityZFiltered;	
		OperationControlData.stForwardXMC1ToOC.MO_origE_IMUX					:=			XMCData.stFromXMC1ToMC.EM_origE_IMUX;		
		OperationControlData.stForwardXMC1ToOC.MO_origE_IMUY					:=			XMCData.stFromXMC1ToMC.EM_origE_IMUY;		
		OperationControlData.stForwardXMC1ToOC.MO_origE_IMUZ					:=			XMCData.stFromXMC1ToMC.EM_origE_IMUZ;		
		OperationControlData.stForwardXMC1ToOC.MO_origE_PressureBox				:=			XMCData.stFromXMC1ToMC.EM_origE_PressureBox;	
		OperationControlData.stForwardXMC1ToOC.MO_origE_TemperatureBox			:=			XMCData.stFromXMC1ToMC.EM_origE_TemperatureBox;		
		OperationControlData.stForwardXMC1ToOC.MO_origE_TemperatureGuid			:=			XMCData.stFromXMC1ToMC.EM_origE_TemperatureGuid;	
		OperationControlData.stForwardXMC1ToOC.MO_origE_TemperatureLev0			:=			XMCData.stFromXMC1ToMC.EM_origE_TemperatureLev0;	
		OperationControlData.stForwardXMC1ToOC.MO_origE_TemperatureLev1			:=			XMCData.stFromXMC1ToMC.EM_origE_TemperatureLev1;	
		//System Status
		OperationControlData.stForwardXMC1ToOC.MO_origE_ErrBits					:=			XMCData.stFromXMC1ToMC.EM_origE_ErrBits;	
		OperationControlData.stForwardXMC1ToOC.MO_origE_SafetyCounter			:=			XMCData.stFromXMC1ToMC.EM_origE_SafetyCounter;		
		OperationControlData.stForwardXMC1ToOC.MO_origE_State					:=			XMCData.stFromXMC1ToMC.EM_origE_State;		
		OperationControlData.stForwardXMC1ToOC.MO_origE_Timestamp				:=			XMCData.stFromXMC1ToMC.EM_origE_Timestamp;		
		OperationControlData.stForwardXMC1ToOC.MO_origE_WarnBits				:=			XMCData.stFromXMC1ToMC.EM_origE_WarnBits;		
		OperationControlData.stForwardXMC1ToOC.MO_origE_LoggingCounterIn		:=			XMCData.stFromXMC1ToMC.EM_origE_LoggingCounterIn;		
		OperationControlData.stForwardXMC1ToOC.MO_origE_LoggingCounterSize		:=			XMCData.stFromXMC1ToMC.EM_origE_LoggingCounterSize;		
		OperationControlData.stForwardXMC1ToOC.MO_origE_LoggingCounterBuf0		:=			XMCData.stFromXMC1ToMC.EM_origE_LoggingCounterBuf0;	
		OperationControlData.stForwardXMC1ToOC.MO_origE_LoggingCounterBuf1		:=			XMCData.stFromXMC1ToMC.EM_origE_LoggingCounterBuf1;	
		OperationControlData.stForwardXMC1ToOC.MO_origE_LoggingCounterBuf2		:=			XMCData.stFromXMC1ToMC.EM_origE_LoggingCounterBuf2;	
		OperationControlData.stForwardXMC1ToOC.MO_origE_LoggingCounterBuf3		:=			XMCData.stFromXMC1ToMC.EM_origE_LoggingCounterBuf3;	
		OperationControlData.stForwardXMC1ToOC.MO_origE_LoggingCounterBuf4		:=			XMCData.stFromXMC1ToMC.EM_origE_LoggingCounterBuf4;	
		OperationControlData.stForwardXMC1ToOC.MO_origE_LoggingCounterBuf5		:=			XMCData.stFromXMC1ToMC.EM_origE_LoggingCounterBuf5;	
		OperationControlData.stForwardXMC1ToOC.MO_origE_LoggingCounterBuf6		:=			XMCData.stFromXMC1ToMC.EM_origE_LoggingCounterBuf6;	
		OperationControlData.stForwardXMC1ToOC.MO_origE_LoggingCounterBuf7		:=			XMCData.stFromXMC1ToMC.EM_origE_LoggingCounterBuf7;	
		OperationControlData.stForwardXMC1ToOC.MO_origE_LoggingCounterBuf8		:=			XMCData.stFromXMC1ToMC.EM_origE_LoggingCounterBuf8;
		OperationControlData.stForwardXMC1ToOC.MO_origE_LoggingCounterBuf9		:=			XMCData.stFromXMC1ToMC.EM_origE_LoggingCounterBuf9;			
		//Levitation
		OperationControlData.stForwardXMC1ToOC.MO_origE_LevEstimatedFlux0[0]		:=			XMCData.stFromXMC1ToMC.EM_origE_LevEstimatedFlux0[0];
		OperationControlData.stForwardXMC1ToOC.MO_origE_LevEstimatedFlux0[1]		:=			XMCData.stFromXMC1ToMC.EM_origE_LevEstimatedFlux0[1];		
		OperationControlData.stForwardXMC1ToOC.MO_origE_LevEstimatedFlux1[0]       :=			XMCData.stFromXMC1ToMC.EM_origE_LevEstimatedFlux1[0]; 
		OperationControlData.stForwardXMC1ToOC.MO_origE_LevEstimatedFlux1[1]       :=			XMCData.stFromXMC1ToMC.EM_origE_LevEstimatedFlux1[1];      
		OperationControlData.stForwardXMC1ToOC.MO_origE_LevEstimatedCurrent     :=			XMCData.stFromXMC1ToMC.EM_origE_LevEstimatedCurrent;       
		OperationControlData.stForwardXMC1ToOC.MO_origE_LevEstimatedResistance  :=			XMCData.stFromXMC1ToMC.EM_origE_LevEstimatedResistance;       
		OperationControlData.stForwardXMC1ToOC.MO_origE_LevIntegratedControlError :=		XMCData.stFromXMC1ToMC.EM_origE_LevIntegratedControlError;       
		OperationControlData.stForwardXMC1ToOC.MO_origE_LevReferenceVoltage     :=			XMCData.stFromXMC1ToMC.EM_origE_LevReferenceVoltage;       
		//Guidance                                 
		OperationControlData.stForwardXMC1ToOC.MO_origE_GuidEstimatedFlux0[0]      :=			XMCData.stFromXMC1ToMC.EM_origE_GuidEstimatedFlux0[0]; 
		OperationControlData.stForwardXMC1ToOC.MO_origE_GuidEstimatedFlux0[1]      :=			XMCData.stFromXMC1ToMC.EM_origE_GuidEstimatedFlux0[1];      
		OperationControlData.stForwardXMC1ToOC.MO_origE_GuidEstimatedFlux1[0]		:=			XMCData.stFromXMC1ToMC.EM_origE_GuidEstimatedFlux1[0];
		OperationControlData.stForwardXMC1ToOC.MO_origE_GuidEstimatedFlux1[1]		:=			XMCData.stFromXMC1ToMC.EM_origE_GuidEstimatedFlux1[1];		
		OperationControlData.stForwardXMC1ToOC.MO_origE_GuidEstimatedCurrent	:=			XMCData.stFromXMC1ToMC.EM_origE_GuidEstimatedCurrent;		
		OperationControlData.stForwardXMC1ToOC.MO_origE_GuidEstimatedResistance	:=			XMCData.stFromXMC1ToMC.EM_origE_GuidEstimatedResistance;	
		OperationControlData.stForwardXMC1ToOC.MO_origE_GuidIntegratedControlError :=		XMCData.stFromXMC1ToMC.EM_origE_GuidIntegratedControlError;		
		OperationControlData.stForwardXMC1ToOC.MO_origE_GuidReferenceVoltage	:=			XMCData.stFromXMC1ToMC.EM_origE_GuidReferenceVoltage;		
	
	//XMC2
		OperationControlData.stForwardXMC2ToOC.MO_origE_CurrentGuid				:=			XMCData.stFromXMC2ToMC.EM_origE_CurrentGuid;			
		OperationControlData.stForwardXMC2ToOC.MO_origE_CurrentLev				:=			XMCData.stFromXMC2ToMC.EM_origE_CurrentLev;		
		OperationControlData.stForwardXMC2ToOC.MO_origE_DistanceRawLev11		:=			XMCData.stFromXMC2ToMC.EM_origE_DistanceRawLev11;		
		OperationControlData.stForwardXMC2ToOC.MO_origE_DistanceRawLev12		:=			XMCData.stFromXMC2ToMC.EM_origE_DistanceRawLev12;		
		OperationControlData.stForwardXMC2ToOC.MO_origE_DistanceRawLev21		:=			XMCData.stFromXMC2ToMC.EM_origE_DistanceRawLev21;		
		OperationControlData.stForwardXMC2ToOC.MO_origE_DistanceRawLev22		:=			XMCData.stFromXMC2ToMC.EM_origE_DistanceRawLev22;		
		OperationControlData.stForwardXMC2ToOC.MO_origE_DistanceRawGuid11		:=			XMCData.stFromXMC2ToMC.EM_origE_DistanceRawGuid11;		
		OperationControlData.stForwardXMC2ToOC.MO_origE_DistanceRawGuid12		:=			XMCData.stFromXMC2ToMC.EM_origE_DistanceRawGuid12;		
		OperationControlData.stForwardXMC2ToOC.MO_origE_DistanceGuidanceFiltered	:=			XMCData.stFromXMC2ToMC.EM_origE_DistanceGuidanceFiltered;		
		OperationControlData.stForwardXMC2ToOC.MO_origE_DistanceLevitationFiltered		:=			XMCData.stFromXMC2ToMC.EM_origE_DistanceLevitationFiltered;	
		OperationControlData.stForwardXMC2ToOC.MO_origE_VelocityZFiltered		:=			XMCData.stFromXMC2ToMC.EM_origE_VelocityZFiltered;	
		OperationControlData.stForwardXMC2ToOC.MO_origE_IMUX					:=			XMCData.stFromXMC2ToMC.EM_origE_IMUX;		
		OperationControlData.stForwardXMC2ToOC.MO_origE_IMUY					:=			XMCData.stFromXMC2ToMC.EM_origE_IMUY;		
		OperationControlData.stForwardXMC2ToOC.MO_origE_IMUZ					:=			XMCData.stFromXMC2ToMC.EM_origE_IMUZ;		
		OperationControlData.stForwardXMC2ToOC.MO_origE_PressureBox				:=			XMCData.stFromXMC2ToMC.EM_origE_PressureBox;	
		OperationControlData.stForwardXMC2ToOC.MO_origE_TemperatureBox			:=			XMCData.stFromXMC2ToMC.EM_origE_TemperatureBox;		
		OperationControlData.stForwardXMC2ToOC.MO_origE_TemperatureGuid			:=			XMCData.stFromXMC2ToMC.EM_origE_TemperatureGuid;	
		OperationControlData.stForwardXMC2ToOC.MO_origE_TemperatureLev0			:=			XMCData.stFromXMC2ToMC.EM_origE_TemperatureLev0;	
		OperationControlData.stForwardXMC2ToOC.MO_origE_TemperatureLev1			:=			XMCData.stFromXMC2ToMC.EM_origE_TemperatureLev1;	
		//System Status
		OperationControlData.stForwardXMC2ToOC.MO_origE_ErrBits					:=			XMCData.stFromXMC2ToMC.EM_origE_ErrBits;	
		OperationControlData.stForwardXMC2ToOC.MO_origE_SafetyCounter			:=			XMCData.stFromXMC2ToMC.EM_origE_SafetyCounter;		
		OperationControlData.stForwardXMC2ToOC.MO_origE_State					:=			XMCData.stFromXMC2ToMC.EM_origE_State;		
		OperationControlData.stForwardXMC2ToOC.MO_origE_Timestamp				:=			XMCData.stFromXMC2ToMC.EM_origE_Timestamp;		
		OperationControlData.stForwardXMC2ToOC.MO_origE_WarnBits				:=			XMCData.stFromXMC2ToMC.EM_origE_WarnBits;		
		OperationControlData.stForwardXMC2ToOC.MO_origE_LoggingCounterIn		:=			XMCData.stFromXMC2ToMC.EM_origE_LoggingCounterIn;		
		OperationControlData.stForwardXMC2ToOC.MO_origE_LoggingCounterSize		:=			XMCData.stFromXMC2ToMC.EM_origE_LoggingCounterSize;		
		OperationControlData.stForwardXMC1ToOC.MO_origE_LoggingCounterBuf0		:=			XMCData.stFromXMC1ToMC.EM_origE_LoggingCounterBuf0;	
		OperationControlData.stForwardXMC1ToOC.MO_origE_LoggingCounterBuf1		:=			XMCData.stFromXMC1ToMC.EM_origE_LoggingCounterBuf1;	
		OperationControlData.stForwardXMC1ToOC.MO_origE_LoggingCounterBuf2		:=			XMCData.stFromXMC1ToMC.EM_origE_LoggingCounterBuf2;	
		OperationControlData.stForwardXMC1ToOC.MO_origE_LoggingCounterBuf3		:=			XMCData.stFromXMC1ToMC.EM_origE_LoggingCounterBuf3;	
		OperationControlData.stForwardXMC1ToOC.MO_origE_LoggingCounterBuf4		:=			XMCData.stFromXMC1ToMC.EM_origE_LoggingCounterBuf4;	
		OperationControlData.stForwardXMC1ToOC.MO_origE_LoggingCounterBuf5		:=			XMCData.stFromXMC1ToMC.EM_origE_LoggingCounterBuf5;	
		OperationControlData.stForwardXMC1ToOC.MO_origE_LoggingCounterBuf6		:=			XMCData.stFromXMC1ToMC.EM_origE_LoggingCounterBuf6;	
		OperationControlData.stForwardXMC1ToOC.MO_origE_LoggingCounterBuf7		:=			XMCData.stFromXMC1ToMC.EM_origE_LoggingCounterBuf7;	
		OperationControlData.stForwardXMC1ToOC.MO_origE_LoggingCounterBuf8		:=			XMCData.stFromXMC1ToMC.EM_origE_LoggingCounterBuf8;
		OperationControlData.stForwardXMC1ToOC.MO_origE_LoggingCounterBuf9		:=			XMCData.stFromXMC1ToMC.EM_origE_LoggingCounterBuf9;		
		//Levitation
		OperationControlData.stForwardXMC2ToOC.MO_origE_LevEstimatedFlux0[0]		:=			XMCData.stFromXMC2ToMC.EM_origE_LevEstimatedFlux0[0];
		OperationControlData.stForwardXMC2ToOC.MO_origE_LevEstimatedFlux0[1]		:=			XMCData.stFromXMC2ToMC.EM_origE_LevEstimatedFlux0[1];		
		OperationControlData.stForwardXMC2ToOC.MO_origE_LevEstimatedFlux1[0]       :=			XMCData.stFromXMC2ToMC.EM_origE_LevEstimatedFlux1[0]; 
		OperationControlData.stForwardXMC2ToOC.MO_origE_LevEstimatedFlux1[1]       :=			XMCData.stFromXMC2ToMC.EM_origE_LevEstimatedFlux1[1];       
		OperationControlData.stForwardXMC2ToOC.MO_origE_LevEstimatedCurrent     :=			XMCData.stFromXMC2ToMC.EM_origE_LevEstimatedCurrent;       
		OperationControlData.stForwardXMC2ToOC.MO_origE_LevEstimatedResistance  :=			XMCData.stFromXMC2ToMC.EM_origE_LevEstimatedResistance;       
		OperationControlData.stForwardXMC2ToOC.MO_origE_LevIntegratedControlError :=		XMCData.stFromXMC2ToMC.EM_origE_LevIntegratedControlError;       
		OperationControlData.stForwardXMC2ToOC.MO_origE_LevReferenceVoltage     :=			XMCData.stFromXMC2ToMC.EM_origE_LevReferenceVoltage;       
		//Guidance                                 
		OperationControlData.stForwardXMC2ToOC.MO_origE_GuidEstimatedFlux0[0]      :=			XMCData.stFromXMC2ToMC.EM_origE_GuidEstimatedFlux0[0]; 
		OperationControlData.stForwardXMC2ToOC.MO_origE_GuidEstimatedFlux0[1]      :=			XMCData.stFromXMC2ToMC.EM_origE_GuidEstimatedFlux0[1];      
		OperationControlData.stForwardXMC2ToOC.MO_origE_GuidEstimatedFlux1[0]		:=			XMCData.stFromXMC2ToMC.EM_origE_GuidEstimatedFlux1[0];
		OperationControlData.stForwardXMC2ToOC.MO_origE_GuidEstimatedFlux1[1]		:=			XMCData.stFromXMC2ToMC.EM_origE_GuidEstimatedFlux1[1];	
		OperationControlData.stForwardXMC2ToOC.MO_origE_GuidEstimatedCurrent	:=			XMCData.stFromXMC2ToMC.EM_origE_GuidEstimatedCurrent;		
		OperationControlData.stForwardXMC2ToOC.MO_origE_GuidEstimatedResistance	:=			XMCData.stFromXMC2ToMC.EM_origE_GuidEstimatedResistance;	
		OperationControlData.stForwardXMC2ToOC.MO_origE_GuidIntegratedControlError :=		XMCData.stFromXMC2ToMC.EM_origE_GuidIntegratedControlError;		
		OperationControlData.stForwardXMC2ToOC.MO_origE_GuidReferenceVoltage	:=			XMCData.stFromXMC2ToMC.EM_origE_GuidReferenceVoltage;		

	//XMC3
		OperationControlData.stForwardXMC3ToOC.MO_origE_CurrentGuid				:=			XMCData.stFromXMC3ToMC.EM_origE_CurrentGuid;			
		OperationControlData.stForwardXMC3ToOC.MO_origE_CurrentLev				:=			XMCData.stFromXMC3ToMC.EM_origE_CurrentLev;		
		OperationControlData.stForwardXMC3ToOC.MO_origE_DistanceRawLev11		:=			XMCData.stFromXMC3ToMC.EM_origE_DistanceRawLev11;		
		OperationControlData.stForwardXMC3ToOC.MO_origE_DistanceRawLev12		:=			XMCData.stFromXMC3ToMC.EM_origE_DistanceRawLev12;		
		OperationControlData.stForwardXMC3ToOC.MO_origE_DistanceRawLev21		:=			XMCData.stFromXMC3ToMC.EM_origE_DistanceRawLev21;		
		OperationControlData.stForwardXMC3ToOC.MO_origE_DistanceRawLev22		:=			XMCData.stFromXMC3ToMC.EM_origE_DistanceRawLev22;		
		OperationControlData.stForwardXMC3ToOC.MO_origE_DistanceRawGuid11		:=			XMCData.stFromXMC3ToMC.EM_origE_DistanceRawGuid11;		
		OperationControlData.stForwardXMC3ToOC.MO_origE_DistanceRawGuid12		:=			XMCData.stFromXMC3ToMC.EM_origE_DistanceRawGuid12;		
		OperationControlData.stForwardXMC3ToOC.MO_origE_DistanceGuidanceFiltered	:=			XMCData.stFromXMC3ToMC.EM_origE_DistanceGuidanceFiltered;		
		OperationControlData.stForwardXMC3ToOC.MO_origE_DistanceLevitationFiltered		:=			XMCData.stFromXMC3ToMC.EM_origE_DistanceLevitationFiltered;	
		OperationControlData.stForwardXMC3ToOC.MO_origE_VelocityZFiltered		:=			XMCData.stFromXMC3ToMC.EM_origE_VelocityZFiltered;	
		OperationControlData.stForwardXMC3ToOC.MO_origE_IMUX					:=			XMCData.stFromXMC3ToMC.EM_origE_IMUX;		
		OperationControlData.stForwardXMC3ToOC.MO_origE_IMUY					:=			XMCData.stFromXMC3ToMC.EM_origE_IMUY;		
		OperationControlData.stForwardXMC3ToOC.MO_origE_IMUZ					:=			XMCData.stFromXMC3ToMC.EM_origE_IMUZ;		
		OperationControlData.stForwardXMC3ToOC.MO_origE_PressureBox				:=			XMCData.stFromXMC3ToMC.EM_origE_PressureBox;	
		OperationControlData.stForwardXMC3ToOC.MO_origE_TemperatureBox			:=			XMCData.stFromXMC3ToMC.EM_origE_TemperatureBox;		
		OperationControlData.stForwardXMC3ToOC.MO_origE_TemperatureGuid			:=			XMCData.stFromXMC3ToMC.EM_origE_TemperatureGuid;	
		OperationControlData.stForwardXMC3ToOC.MO_origE_TemperatureLev0			:=			XMCData.stFromXMC3ToMC.EM_origE_TemperatureLev0;	
		OperationControlData.stForwardXMC3ToOC.MO_origE_TemperatureLev1			:=			XMCData.stFromXMC3ToMC.EM_origE_TemperatureLev1;	
		//System Status
		OperationControlData.stForwardXMC3ToOC.MO_origE_ErrBits					:=			XMCData.stFromXMC3ToMC.EM_origE_ErrBits;	
		OperationControlData.stForwardXMC3ToOC.MO_origE_SafetyCounter			:=			XMCData.stFromXMC3ToMC.EM_origE_SafetyCounter;		
		OperationControlData.stForwardXMC3ToOC.MO_origE_State					:=			XMCData.stFromXMC3ToMC.EM_origE_State;		
		OperationControlData.stForwardXMC3ToOC.MO_origE_Timestamp				:=			XMCData.stFromXMC3ToMC.EM_origE_Timestamp;		
		OperationControlData.stForwardXMC3ToOC.MO_origE_WarnBits				:=			XMCData.stFromXMC3ToMC.EM_origE_WarnBits;		
		OperationControlData.stForwardXMC3ToOC.MO_origE_LoggingCounterIn		:=			XMCData.stFromXMC3ToMC.EM_origE_LoggingCounterIn;		
		OperationControlData.stForwardXMC3ToOC.MO_origE_LoggingCounterSize		:=			XMCData.stFromXMC3ToMC.EM_origE_LoggingCounterSize;		
		OperationControlData.stForwardXMC1ToOC.MO_origE_LoggingCounterBuf0		:=			XMCData.stFromXMC1ToMC.EM_origE_LoggingCounterBuf0;	
		OperationControlData.stForwardXMC1ToOC.MO_origE_LoggingCounterBuf1		:=			XMCData.stFromXMC1ToMC.EM_origE_LoggingCounterBuf1;	
		OperationControlData.stForwardXMC1ToOC.MO_origE_LoggingCounterBuf2		:=			XMCData.stFromXMC1ToMC.EM_origE_LoggingCounterBuf2;	
		OperationControlData.stForwardXMC1ToOC.MO_origE_LoggingCounterBuf3		:=			XMCData.stFromXMC1ToMC.EM_origE_LoggingCounterBuf3;	
		OperationControlData.stForwardXMC1ToOC.MO_origE_LoggingCounterBuf4		:=			XMCData.stFromXMC1ToMC.EM_origE_LoggingCounterBuf4;	
		OperationControlData.stForwardXMC1ToOC.MO_origE_LoggingCounterBuf5		:=			XMCData.stFromXMC1ToMC.EM_origE_LoggingCounterBuf5;	
		OperationControlData.stForwardXMC1ToOC.MO_origE_LoggingCounterBuf6		:=			XMCData.stFromXMC1ToMC.EM_origE_LoggingCounterBuf6;	
		OperationControlData.stForwardXMC1ToOC.MO_origE_LoggingCounterBuf7		:=			XMCData.stFromXMC1ToMC.EM_origE_LoggingCounterBuf7;	
		OperationControlData.stForwardXMC1ToOC.MO_origE_LoggingCounterBuf8		:=			XMCData.stFromXMC1ToMC.EM_origE_LoggingCounterBuf8;
		OperationControlData.stForwardXMC1ToOC.MO_origE_LoggingCounterBuf9		:=			XMCData.stFromXMC1ToMC.EM_origE_LoggingCounterBuf9;		
		//Levitation
		OperationControlData.stForwardXMC3ToOC.MO_origE_LevEstimatedFlux0[0]		:=			XMCData.stFromXMC3ToMC.EM_origE_LevEstimatedFlux0[0];
		OperationControlData.stForwardXMC3ToOC.MO_origE_LevEstimatedFlux0[1]		:=			XMCData.stFromXMC3ToMC.EM_origE_LevEstimatedFlux0[1];		
		OperationControlData.stForwardXMC3ToOC.MO_origE_LevEstimatedFlux1[0]       :=			XMCData.stFromXMC3ToMC.EM_origE_LevEstimatedFlux1[0]; 
		OperationControlData.stForwardXMC3ToOC.MO_origE_LevEstimatedFlux1[1]       :=			XMCData.stFromXMC3ToMC.EM_origE_LevEstimatedFlux1[1];       
		OperationControlData.stForwardXMC3ToOC.MO_origE_LevEstimatedCurrent     :=			XMCData.stFromXMC3ToMC.EM_origE_LevEstimatedCurrent;       
		OperationControlData.stForwardXMC3ToOC.MO_origE_LevEstimatedResistance  :=			XMCData.stFromXMC3ToMC.EM_origE_LevEstimatedResistance;       
		OperationControlData.stForwardXMC3ToOC.MO_origE_LevIntegratedControlError :=		XMCData.stFromXMC3ToMC.EM_origE_LevIntegratedControlError;       
		OperationControlData.stForwardXMC3ToOC.MO_origE_LevReferenceVoltage     :=			XMCData.stFromXMC3ToMC.EM_origE_LevReferenceVoltage;       
		//Guidance                                 
		OperationControlData.stForwardXMC3ToOC.MO_origE_GuidEstimatedFlux0[0]      :=			XMCData.stFromXMC3ToMC.EM_origE_GuidEstimatedFlux0[0]; 
		OperationControlData.stForwardXMC3ToOC.MO_origE_GuidEstimatedFlux0[1]      :=			XMCData.stFromXMC3ToMC.EM_origE_GuidEstimatedFlux0[1];      
		OperationControlData.stForwardXMC3ToOC.MO_origE_GuidEstimatedFlux1[0]		:=			XMCData.stFromXMC3ToMC.EM_origE_GuidEstimatedFlux1[0];
		OperationControlData.stForwardXMC3ToOC.MO_origE_GuidEstimatedFlux1[1]		:=			XMCData.stFromXMC3ToMC.EM_origE_GuidEstimatedFlux1[1];		
		OperationControlData.stForwardXMC3ToOC.MO_origE_GuidEstimatedCurrent	:=			XMCData.stFromXMC3ToMC.EM_origE_GuidEstimatedCurrent;		
		OperationControlData.stForwardXMC3ToOC.MO_origE_GuidEstimatedResistance	:=			XMCData.stFromXMC3ToMC.EM_origE_GuidEstimatedResistance;	
		OperationControlData.stForwardXMC3ToOC.MO_origE_GuidIntegratedControlError :=		XMCData.stFromXMC3ToMC.EM_origE_GuidIntegratedControlError;		
		OperationControlData.stForwardXMC3ToOC.MO_origE_GuidReferenceVoltage	:=			XMCData.stFromXMC3ToMC.EM_origE_GuidReferenceVoltage;	

	//XMC4
		OperationControlData.stForwardXMC4ToOC.MO_origE_CurrentGuid				:=			XMCData.stFromXMC4ToMC.EM_origE_CurrentGuid;			
		OperationControlData.stForwardXMC4ToOC.MO_origE_CurrentLev				:=			XMCData.stFromXMC4ToMC.EM_origE_CurrentLev;		
		OperationControlData.stForwardXMC4ToOC.MO_origE_DistanceRawLev11		:=			XMCData.stFromXMC4ToMC.EM_origE_DistanceRawLev11;		
		OperationControlData.stForwardXMC4ToOC.MO_origE_DistanceRawLev12		:=			XMCData.stFromXMC4ToMC.EM_origE_DistanceRawLev12;		
		OperationControlData.stForwardXMC4ToOC.MO_origE_DistanceRawLev21		:=			XMCData.stFromXMC4ToMC.EM_origE_DistanceRawLev21;		
		OperationControlData.stForwardXMC4ToOC.MO_origE_DistanceRawLev22		:=			XMCData.stFromXMC4ToMC.EM_origE_DistanceRawLev22;		
		OperationControlData.stForwardXMC4ToOC.MO_origE_DistanceRawGuid11		:=			XMCData.stFromXMC4ToMC.EM_origE_DistanceRawGuid11;		
		OperationControlData.stForwardXMC4ToOC.MO_origE_DistanceRawGuid12		:=			XMCData.stFromXMC4ToMC.EM_origE_DistanceRawGuid12;		
		OperationControlData.stForwardXMC4ToOC.MO_origE_DistanceGuidanceFiltered	:=			XMCData.stFromXMC4ToMC.EM_origE_DistanceGuidanceFiltered;		
		OperationControlData.stForwardXMC4ToOC.MO_origE_DistanceLevitationFiltered		:=			XMCData.stFromXMC4ToMC.EM_origE_DistanceLevitationFiltered;	
		OperationControlData.stForwardXMC4ToOC.MO_origE_VelocityZFiltered		:=			XMCData.stFromXMC4ToMC.EM_origE_VelocityZFiltered;	
		OperationControlData.stForwardXMC4ToOC.MO_origE_IMUX					:=			XMCData.stFromXMC4ToMC.EM_origE_IMUX;		
		OperationControlData.stForwardXMC4ToOC.MO_origE_IMUY					:=			XMCData.stFromXMC4ToMC.EM_origE_IMUY;		
		OperationControlData.stForwardXMC4ToOC.MO_origE_IMUZ					:=			XMCData.stFromXMC4ToMC.EM_origE_IMUZ;		
		OperationControlData.stForwardXMC4ToOC.MO_origE_PressureBox				:=			XMCData.stFromXMC4ToMC.EM_origE_PressureBox;	
		OperationControlData.stForwardXMC4ToOC.MO_origE_TemperatureBox			:=			XMCData.stFromXMC4ToMC.EM_origE_TemperatureBox;		
		OperationControlData.stForwardXMC4ToOC.MO_origE_TemperatureGuid			:=			XMCData.stFromXMC4ToMC.EM_origE_TemperatureGuid;	
		OperationControlData.stForwardXMC4ToOC.MO_origE_TemperatureLev0			:=			XMCData.stFromXMC4ToMC.EM_origE_TemperatureLev0;	
		OperationControlData.stForwardXMC4ToOC.MO_origE_TemperatureLev1			:=			XMCData.stFromXMC4ToMC.EM_origE_TemperatureLev1;	
		//System Status
		OperationControlData.stForwardXMC4ToOC.MO_origE_ErrBits					:=			XMCData.stFromXMC4ToMC.EM_origE_ErrBits;	
		OperationControlData.stForwardXMC4ToOC.MO_origE_SafetyCounter			:=			XMCData.stFromXMC4ToMC.EM_origE_SafetyCounter;		
		OperationControlData.stForwardXMC4ToOC.MO_origE_State					:=			XMCData.stFromXMC4ToMC.EM_origE_State;		
		OperationControlData.stForwardXMC4ToOC.MO_origE_Timestamp				:=			XMCData.stFromXMC4ToMC.EM_origE_Timestamp;		
		OperationControlData.stForwardXMC4ToOC.MO_origE_WarnBits				:=			XMCData.stFromXMC4ToMC.EM_origE_WarnBits;		
		OperationControlData.stForwardXMC4ToOC.MO_origE_LoggingCounterIn		:=			XMCData.stFromXMC4ToMC.EM_origE_LoggingCounterIn;		
		OperationControlData.stForwardXMC4ToOC.MO_origE_LoggingCounterSize		:=			XMCData.stFromXMC4ToMC.EM_origE_LoggingCounterSize;		
		OperationControlData.stForwardXMC1ToOC.MO_origE_LoggingCounterBuf0		:=			XMCData.stFromXMC1ToMC.EM_origE_LoggingCounterBuf0;	
		OperationControlData.stForwardXMC1ToOC.MO_origE_LoggingCounterBuf1		:=			XMCData.stFromXMC1ToMC.EM_origE_LoggingCounterBuf1;	
		OperationControlData.stForwardXMC1ToOC.MO_origE_LoggingCounterBuf2		:=			XMCData.stFromXMC1ToMC.EM_origE_LoggingCounterBuf2;	
		OperationControlData.stForwardXMC1ToOC.MO_origE_LoggingCounterBuf3		:=			XMCData.stFromXMC1ToMC.EM_origE_LoggingCounterBuf3;	
		OperationControlData.stForwardXMC1ToOC.MO_origE_LoggingCounterBuf4		:=			XMCData.stFromXMC1ToMC.EM_origE_LoggingCounterBuf4;	
		OperationControlData.stForwardXMC1ToOC.MO_origE_LoggingCounterBuf5		:=			XMCData.stFromXMC1ToMC.EM_origE_LoggingCounterBuf5;	
		OperationControlData.stForwardXMC1ToOC.MO_origE_LoggingCounterBuf6		:=			XMCData.stFromXMC1ToMC.EM_origE_LoggingCounterBuf6;	
		OperationControlData.stForwardXMC1ToOC.MO_origE_LoggingCounterBuf7		:=			XMCData.stFromXMC1ToMC.EM_origE_LoggingCounterBuf7;	
		OperationControlData.stForwardXMC1ToOC.MO_origE_LoggingCounterBuf8		:=			XMCData.stFromXMC1ToMC.EM_origE_LoggingCounterBuf8;
		OperationControlData.stForwardXMC1ToOC.MO_origE_LoggingCounterBuf9		:=			XMCData.stFromXMC1ToMC.EM_origE_LoggingCounterBuf9;		
		//Levitation
		OperationControlData.stForwardXMC4ToOC.MO_origE_LevEstimatedFlux0[0]		:=			XMCData.stFromXMC4ToMC.EM_origE_LevEstimatedFlux0[0];
		OperationControlData.stForwardXMC4ToOC.MO_origE_LevEstimatedFlux0[1]		:=			XMCData.stFromXMC4ToMC.EM_origE_LevEstimatedFlux0[1];		
		OperationControlData.stForwardXMC4ToOC.MO_origE_LevEstimatedFlux1[0]       :=			XMCData.stFromXMC4ToMC.EM_origE_LevEstimatedFlux1[0]; 
		OperationControlData.stForwardXMC4ToOC.MO_origE_LevEstimatedFlux1[1]       :=			XMCData.stFromXMC4ToMC.EM_origE_LevEstimatedFlux1[1];       
		OperationControlData.stForwardXMC4ToOC.MO_origE_LevEstimatedCurrent     :=			XMCData.stFromXMC4ToMC.EM_origE_LevEstimatedCurrent;       
		OperationControlData.stForwardXMC4ToOC.MO_origE_LevEstimatedResistance  :=			XMCData.stFromXMC4ToMC.EM_origE_LevEstimatedResistance;       
		OperationControlData.stForwardXMC4ToOC.MO_origE_LevIntegratedControlError :=		XMCData.stFromXMC4ToMC.EM_origE_LevIntegratedControlError;       
		OperationControlData.stForwardXMC4ToOC.MO_origE_LevReferenceVoltage     :=			XMCData.stFromXMC4ToMC.EM_origE_LevReferenceVoltage;       
		//Guidance                                 
		OperationControlData.stForwardXMC4ToOC.MO_origE_GuidEstimatedFlux0[0]      :=			XMCData.stFromXMC4ToMC.EM_origE_GuidEstimatedFlux0[0]; 
		OperationControlData.stForwardXMC4ToOC.MO_origE_GuidEstimatedFlux0[1]      :=			XMCData.stFromXMC4ToMC.EM_origE_GuidEstimatedFlux0[1];      
		OperationControlData.stForwardXMC4ToOC.MO_origE_GuidEstimatedFlux1[0]		:=			XMCData.stFromXMC4ToMC.EM_origE_GuidEstimatedFlux1[0];
		OperationControlData.stForwardXMC4ToOC.MO_origE_GuidEstimatedFlux1[1]		:=			XMCData.stFromXMC4ToMC.EM_origE_GuidEstimatedFlux1[1];		
		OperationControlData.stForwardXMC4ToOC.MO_origE_GuidEstimatedCurrent	:=			XMCData.stFromXMC4ToMC.EM_origE_GuidEstimatedCurrent;		
		OperationControlData.stForwardXMC4ToOC.MO_origE_GuidEstimatedResistance	:=			XMCData.stFromXMC4ToMC.EM_origE_GuidEstimatedResistance;	
		OperationControlData.stForwardXMC4ToOC.MO_origE_GuidIntegratedControlError :=		XMCData.stFromXMC4ToMC.EM_origE_GuidIntegratedControlError;		
		OperationControlData.stForwardXMC4ToOC.MO_origE_GuidReferenceVoltage	:=			XMCData.stFromXMC4ToMC.EM_origE_GuidReferenceVoltage;
END_METHOD

METHOD doEnableSystems
VAR_INPUT
END_VAR
IF NOT stOperationControlCommands.nOperationMode.0 THEN
	fbServiceModule.eActivationStatus := ActivationStatus.Enabled;
ELSE
	fbServiceModule.eActivationStatus := ActivationStatus.Disabled;
END_IF

IF NOT stOperationControlCommands.nOperationMode.1 THEN
	fbLevitationSystem.eActivationStatus := ActivationStatus.Enabled;
ELSE
	fbLevitationSystem.eActivationStatus := ActivationStatus.Disabled;
END_IF

IF NOT stOperationControlCommands.nOperationMode.2 THEN
	fbGuidanceSystem.eActivationStatus := ActivationStatus.Enabled;
ELSE
	fbGuidanceSystem.eActivationStatus := ActivationStatus.Disabled;
END_IF
END_METHOD

END_PROGRAM

// ---- POUs/FB_ServiceModule.TcPOU
FUNCTION_BLOCK FB_ServiceModule EXTENDS FB_HighLevelSystem
VAR_INPUT
	eState : ServiceModuleSTM;
	//eActivationStatus : ActivationStatus;
END_VAR
VAR
	//Components
	fbDistanceSensor : FB_DistanceSensor;
	fbBoxLED : FB_BoxLED;
	fbRGBLED : FB_RGBLED;
END_VAR

IF eActivationStatus = ActivationStatus.Enabled THEN
	//High Level State Machine
	CASE eState OF
		ServiceModuleSTM.Idling:
				fbDistanceSensor();
				fbRGBLED(eColor:=LEDColor.Off);
				fbBoxLED(eMode:=LEDMode.Off);
	
		ServiceModuleSTM.Waiting:
				fbRGBLED.eColor := LEDColor.Blue;
				fbBoxLED.eMode := LEDMode.SlowFlashing;
				fbDistanceSensor();
				fbRGBLED();
				fbBoxLED();
				
	
		ServiceModuleSTM.Running:
				fbRGBLED.eColor := LEDColor.Green;
				fbBoxLED.eMode := LEDMode.On;
				fbDistanceSensor();
				fbRGBLED();
				fbBoxLED();
	
		ServiceModuleSTM.PostRunning:
				fbRGBLED.eColor := LEDColor.Red;
				fbBoxLED.eMode := LEDMode.Dimmed;
				fbDistanceSensor();
				fbRGBLED();
				fbBoxLED();
	
		ServiceModuleSTM.PreparingForError:
				fbRGBLED.eColor := LEDColor.Red;
				fbBoxLED.eMode := LEDMode.FastFlashing;
				fbRGBLED();
				fbBoxLED();
	END_CASE
END_IF

PROPERTY eCondition : HighLevelCondition
GET
IF eActivationStatus = ActivationStatus.Disabled THEN
	eCondition := HighLevelCondition.SLEEP;
ELSE
	IF fbDistanceSensor.eCondition = SubLevelCondition.RUN AND fbBoxLED.eCondition = SubLevelCondition.RUN AND fbRGBLED.eCondition = SubLevelCondition.RUN THEN
		eCondition := HighLevelCondition.RUN;
	ELSE
		eCondition := HighLevelCondition.INIT;
	END_IF
END_IF
END_GET
END_PROPERTY

PROPERTY fDistance : REAL
GET
fDistance := LREAL_TO_REAL(fbDistanceSensor.fDistance);
END_GET
END_PROPERTY

PROPERTY nErrorID : UDINT
GET
VAR
	nErrorBitsDS : UDINT;
	nErrorBitsBox : UDINT;
	nErrorBitsRGB : UDINT;
END_VAR
nErrorBitsDS := fbDistanceSensor.nErrorID;
nErrorBitsBox:= fbBoxLED.nErrorID;
nErrorBitsRGB := fbRGBLED.nErrorID;

nErrorID.0 := nErrorBitsDS.0;
nErrorID.1 := nErrorBitsDS.1;
nErrorID.2 := nErrorBitsBox.0;
nErrorID.3 := nErrorBitsBox.1;
nErrorID.4 := nErrorBitsRGB.0;
nErrorID.5 := nErrorBitsRGB.1;
nErrorID.6 := nErrorBitsRGB.2;
nErrorID.7 := nErrorBitsRGB.3;
nErrorID.8 := nErrorBitsRGB.4;
nErrorID.9 := nErrorBitsRGB.5;
END_GET
END_PROPERTY

END_FUNCTION_BLOCK

